(* IEC 61131-3 sources: RL_MAR/experiments/results/ablation/Ablation_single_agent_deepseek-ai_DeepSeek-V3.2_20260603_033757, 94 files *)

(* ---- hard_92.st ---- *)
FUNCTION_BLOCK FB_BreakerControlSystem
VAR_INPUT
    B10_1_Trip : BOOL;
    B10_1_Close : BOOL;
    B10_2_Trip : BOOL;
    B10_2_Close : BOOL;
    B10_12_Trip : BOOL;
    B10_12_Close : BOOL;
    B54_Trip : BOOL;
    B54_Close : BOOL;
    B55_Trip : BOOL;
    B55_Close : BOOL;
    B56_Trip : BOOL;
    B56_Close : BOOL;
    B57_Trip : BOOL;
    B57_Close : BOOL;
END_VAR

VAR_OUTPUT
    Point_1a : INT;
    Point_2a : INT;
    Point_3a : INT;
    Point_4a : INT;
    B10_1_Opened : BOOL;
    B10_1_Closed : BOOL;
    B10_2_Opened : BOOL;
    B10_2_Closed : BOOL;
    B10_12_Opened : BOOL;
    B10_12_Closed : BOOL;
    B54_Opened : BOOL;
    B54_Closed : BOOL;
    B55_Opened : BOOL;
    B55_Closed : BOOL;
    B56_Opened : BOOL;
    B56_Closed : BOOL;
    B57_Opened : BOOL;
    B57_Closed : BOOL;
END_VAR

VAR
    SEL86_OUT : INT;
    MOVE89_OUT : INT;
    SEL66_OUT : INT;
    MOVE69_OUT : INT;
    SEL96_OUT : INT;
    MOVE99_OUT : INT;
    SEL106_OUT : INT;
    MOVE109_OUT : INT;
END_VAR

(* Breaker State Transition Logic *)
(* B10_1 State Management *)
IF B10_1_Close THEN
    B10_1_Closed := TRUE;
    B10_1_Opened := FALSE;
ELSIF B10_1_Trip THEN
    B10_1_Closed := FALSE;
    B10_1_Opened := TRUE;
END_IF;

(* B10_2 State Management *)
IF B10_2_Close THEN
    B10_2_Closed := TRUE;
    B10_2_Opened := FALSE;
ELSIF B10_2_Trip THEN
    B10_2_Closed := FALSE;
    B10_2_Opened := TRUE;
END_IF;

(* B10_12 State Management *)
IF B10_12_Close THEN
    B10_12_Closed := TRUE;
    B10_12_Opened := FALSE;
ELSIF B10_12_Trip THEN
    B10_12_Closed := FALSE;
    B10_12_Opened := TRUE;
END_IF;

(* B54 State Management *)
IF B54_Close THEN
    B54_Closed := TRUE;
    B54_Opened := FALSE;
ELSIF B54_Trip THEN
    B54_Closed := FALSE;
    B54_Opened := TRUE;
END_IF;

(* B55 State Management *)
IF B55_Close THEN
    B55_Closed := TRUE;
    B55_Opened := FALSE;
ELSIF B55_Trip THEN
    B55_Closed := FALSE;
    B55_Opened := TRUE;
END_IF;

(* B56 State Management *)
IF B56_Close THEN
    B56_Closed := TRUE;
    B56_Opened := FALSE;
ELSIF B56_Trip THEN
    B56_Closed := FALSE;
    B56_Opened := TRUE;
END_IF;

(* B57 State Management *)
IF B57_Close THEN
    B57_Closed := TRUE;
    B57_Opened := FALSE;
ELSIF B57_Trip THEN
    B57_Closed := FALSE;
    B57_Opened := TRUE;
END_IF;

(* Point_1a Calculation *)
IF B54_Closed AND ((B10_12_Closed AND B10_1_Closed) OR B10_2_Closed) THEN
    Point_1a := 0;
ELSE
    Point_1a := 138;
END_IF;

(* Point_2a Calculation *)
IF B55_Closed AND ((B10_12_Closed AND B10_1_Closed) OR B10_2_Closed) THEN
    Point_2a := 0;
ELSE
    Point_2a := 138;
END_IF;

(* Point_3a Calculation *)
IF B56_Closed AND ((B10_12_Closed AND B10_2_Closed) OR B10_1_Closed) THEN
    Point_3a := 0;
ELSE
    Point_3a := 138;
END_IF;

(* Point_4a Calculation *)
IF B57_Closed AND ((B10_12_Closed AND B10_2_Closed) OR B10_1_Closed) THEN
    Point_4a := 0;
ELSE
    Point_4a := 138;
END_IF;

END_FUNCTION_BLOCK

(* ---- hard_93.st ---- *)
FUNCTION_BLOCK FB_CircuitControl
VAR_INPUT
    Reset_All_CB : BOOL;
    Current_Fault_on_TRSF1 : INT;
    Current_Fault_on_66BUS1 : INT;
END_VAR

VAR_OUTPUT
    Short_Circuit_TRSF1 : BOOL;
    Short_Circuit_66BUS : BOOL;
    Open_CB1_66KV : BOOL;
    Open_CB2_66KV : BOOL;
    Open_CB_TRSF1 : BOOL;
    Open_CB2_22KV : BOOL;
END_VAR

VAR
    Threshold500 : INT := 500;
    Prev_Open_CB2_22KV : BOOL;
    Prev_Open_CB1_66KV : BOOL;
    Prev_Open_CB_TRSF1 : BOOL;
    Temp_Open_CB2_22KV : BOOL;
    Temp_Open_CB1_66KV : BOOL;
    Temp_Open_CB_TRSF1 : BOOL;
END_VAR

(* Short Circuit Detection *)
Short_Circuit_66BUS := (Current_Fault_on_66BUS1 > Threshold500);
Short_Circuit_TRSF1 := (Current_Fault_on_TRSF1 > Threshold500);

(* Save previous states for edge detection and logic *)
Prev_Open_CB2_22KV := Open_CB2_22KV;
Prev_Open_CB1_66KV := Open_CB1_66KV;
Prev_Open_CB_TRSF1 := Open_CB_TRSF1;

(* Initial Reset Condition *)
IF Reset_All_CB THEN
    Open_CB2_22KV := FALSE;
    Open_CB1_66KV := FALSE;
    Open_CB_TRSF1 := FALSE;
    Open_CB2_66KV := TRUE;
    RETURN;
END_IF;

(* Step 1: Initial Open_CB2_22KV Logic *)
Temp_Open_CB2_22KV := FALSE;
IF (Prev_Open_CB2_22KV = FALSE) THEN
    IF ((Open_CB1_66KV AND Open_CB_TRSF1) OR Short_Circuit_66BUS) THEN
        Temp_Open_CB2_22KV := TRUE;
    END_IF;
END_IF;

(* Step 2: Initial Open_CB1_66KV Logic *)
Temp_Open_CB1_66KV := FALSE;
IF (Temp_Open_CB2_22KV = FALSE) THEN
    IF ((Prev_Open_CB1_66KV AND Open_CB_TRSF1) OR Short_Circuit_66BUS) THEN
        Temp_Open_CB1_66KV := TRUE;
    END_IF;
END_IF;

(* Step 3: Initial Open_CB_TRSF1 Logic *)
Temp_Open_CB_TRSF1 := FALSE;
IF (Temp_Open_CB2_22KV = FALSE) THEN
    IF ((Open_CB1_66KV AND Prev_Open_CB_TRSF1) OR Short_Circuit_66BUS) THEN
        Temp_Open_CB_TRSF1 := TRUE;
    END_IF;
END_IF;

(* Step 4: Open_CB2_66KV is always TRUE *)
Open_CB2_66KV := TRUE;

(* Step 5: Update Open_CB2_22KV again *)
IF (Prev_Open_CB2_22KV = FALSE) THEN
    IF ((Open_CB2_66KV AND Open_CB1_66KV AND Open_CB_TRSF1) OR Short_Circuit_TRSF1) THEN
        Temp_Open_CB2_22KV := TRUE;
    END_IF;
END_IF;

(* Step 6: Update Open_CB1_66KV again *)
IF (Temp_Open_CB2_22KV = FALSE) THEN
    IF ((Open_CB2_66KV AND Prev_Open_CB1_66KV AND Open_CB_TRSF1) OR Short_Circuit_TRSF1) THEN
        Temp_Open_CB1_66KV := TRUE;
    END_IF;
END_IF;

(* Step 7: Update Open_CB_TRSF1 again *)
IF (Temp_Open_CB2_22KV = FALSE) THEN
    IF ((Open_CB2_66KV AND Open_CB1_66KV AND Prev_Open_CB_TRSF1) OR Short_Circuit_TRSF1) THEN
        Temp_Open_CB_TRSF1 := TRUE;
    END_IF;
END_IF;

(* Apply final values with anti-rapid switching: only change if new state is TRUE and current is FALSE *)
IF (Temp_Open_CB2_22KV AND (NOT Open_CB2_22KV)) THEN
    Open_CB2_22KV := TRUE;
END_IF;

IF (Temp_Open_CB1_66KV AND (NOT Open_CB1_66KV)) THEN
    Open_CB1_66KV := TRUE;
END_IF;

IF (Temp_Open_CB_TRSF1 AND (NOT Open_CB_TRSF1)) THEN
    Open_CB_TRSF1 := TRUE;
END_IF;

END_FUNCTION_BLOCK

(* ---- hard_94.st ---- *)
FUNCTION_BLOCK FB_AdvancedCircuitBreakerControl
VAR_INPUT
    S_AL1_P_B1 : BOOL;
    S_AL1_P_B2 : BOOL;
    S_AL1_MCB : BOOL;
    MCB_BUSY : BOOL;
    MCB_ERROR : BOOL;
    S_AL1_MCBR : BOOL;
    MCBR_BUSY : BOOL;
    MCBR_ERROR : BOOL;
    S_AL1_P_B3 : BOOL;
    S_AL1_MCB2 : BOOL;
    S_AL1_MCBR2 : BOOL;
END_VAR

VAR_OUTPUT
    E_AL1_B1 : BOOL;
    PUWS_AL1_B1_PLUS : BOOL;
    PUWS_AL1_B1_RIGHT : BOOL;
    PAS_AL1_PLUS : BOOL;
    PAS_AL1_TURN : BOOL;
END_VAR

VAR
    PPAL1 : BOOL := TRUE;
    PP0 : BOOL := TRUE;
    PP1 : BOOL := FALSE;
    PP2 : BOOL := FALSE;
    PP3 : BOOL := FALSE;
    PP4 : BOOL := FALSE;
    MCB : BOOL := TRUE;
    PP5 : BOOL := FALSE;
    PP7 : BOOL := FALSE;
    PPL3 : BOOL := FALSE;
    PPL4 : BOOL := FALSE;
    MCBR : BOOL := TRUE;
    PPL5 : BOOL := FALSE;
    PPL7 : BOOL := FALSE;
    STABLE : BOOL := FALSE;
    MCB_CONTROL : BOOL;
END_VAR

METHOD Main : BOOL
VAR_INST
END_VAR

STABLE := FALSE;

WHILE (STABLE = FALSE) DO
    STABLE := TRUE;

    // PP0 to PP1
    IF (PP0 = TRUE) AND (NOT MCB_CONTROL) AND (PP1 = FALSE) THEN
        PP0 := FALSE;
        PP1 := TRUE;
        STABLE := FALSE;
    END_IF;

    // PP1 to PP2
    IF (PP1 = TRUE) AND S_AL1_P_B1 AND (PP2 = FALSE) THEN
        PP1 := FALSE;
        PP2 := TRUE;
        STABLE := FALSE;
    END_IF;

    // PP2 to PP3
    IF (PP2 = TRUE) AND S_AL1_P_B2 AND (NOT MCB_CONTROL) AND (PP3 = FALSE) THEN
        PP2 := FALSE;
        PP3 := TRUE;
        STABLE := FALSE;
    END_IF;

    // PP3 to PP4
    IF (PP3 = TRUE) AND S_AL1_MCB AND (PP4 = FALSE) AND (PP1 = FALSE) THEN
        PP3 := FALSE;
        PP4 := TRUE;
        PP1 := TRUE;
        STABLE := FALSE;
    END_IF;

    // PP4 to PP5
    IF (PP4 = TRUE) AND (MCB = TRUE) AND MCB_BUSY AND (PP5 = FALSE) THEN
        PP4 := FALSE;
        MCB := FALSE;
        PP5 := TRUE;
        STABLE := FALSE;
    END_IF;

    // PP5 to PP7
    IF (PP5 = TRUE) AND S_AL1_MCB2 AND (PP7 = FALSE) AND (MCB = FALSE) THEN
        PP5 := FALSE;
        PP7 := TRUE;
        MCB := TRUE;
        STABLE := FALSE;
    END_IF;

    // PP7 to End
    IF (PP7 = TRUE) AND S_AL1_P_B3 THEN
        PP7 := FALSE;
        STABLE := FALSE;
    END_IF;

    // PP2 to PPL3
    IF (PP2 = TRUE) AND S_AL1_P_B2 AND MCB_CONTROL AND (PPL3 = FALSE) AND (PP1 = FALSE) THEN
        PP2 := FALSE;
        PPL3 := TRUE;
        PP1 := TRUE;
        STABLE := FALSE;
    END_IF;

    // PPL3 to PPL4
    IF (PPL3 = TRUE) AND S_AL1_MCBR AND (PPL4 = FALSE) THEN
        PPL3 := FALSE;
        PPL4 := TRUE;
        STABLE := FALSE;
    END_IF;

    // PPL4 to PPL5
    IF (PPL4 = TRUE) AND (MCBR = TRUE) AND MCBR_BUSY AND (PPL5 = FALSE) THEN
        PPL4 := FALSE;
        MCBR := FALSE;
        PPL5 := TRUE;
        STABLE := FALSE;
    END_IF;

    // PPL5 to PPL7
    IF (PPL5 = TRUE) AND S_AL1_MCBR2 AND (PPL7 = FALSE) AND (MCBR = FALSE) THEN
        PPL5 := FALSE;
        PPL7 := TRUE;
        MCBR := TRUE;
        STABLE := FALSE;
    END_IF;

    // PPL7 to End
    IF (PPL7 = TRUE) AND S_AL1_P_B3 THEN
        PPL7 := FALSE;
        STABLE := FALSE;
    END_IF;
END_WHILE;

// Output Control
// Set outputs based on active states
IF (PP0 = TRUE) OR (PP1 = TRUE) THEN
    E_AL1_B1 := TRUE;
ELSE
    E_AL1_B1 := FALSE;
END_IF;

IF (PP3 = TRUE) THEN
    MCB_CONTROL := TRUE;
ELSE
    MCB_CONTROL := FALSE;
END_IF;

IF (PPL3 = TRUE) OR (PPL4 = TRUE) THEN
    PAS_AL1_PLUS := TRUE;
    PAS_AL1_TURN := TRUE;
ELSE
    PAS_AL1_PLUS := FALSE;
    PAS_AL1_TURN := FALSE;
END_IF;

IF (PPAL1 = TRUE) OR (PP2 = TRUE) THEN
    PUWS_AL1_B1_PLUS := TRUE;
ELSE
    PUWS_AL1_B1_PLUS := FALSE;
END_IF;

IF (PP2 = TRUE) OR (PP3 = TRUE) OR (PPL3 = TRUE) THEN
    E_AL1_B1 := FALSE;
END_IF;

IF (PP0 = TRUE) OR (PP3 = TRUE) THEN
    MCB_CONTROL := FALSE;
END_IF;

IF (PP0 = TRUE) OR (PP3 = TRUE) OR (PP4 = TRUE) THEN
    PAS_AL1_PLUS := FALSE;
    PAS_AL1_TURN := FALSE;
END_IF;

IF (PPAL1 = TRUE) OR (PP2 = TRUE) THEN
    PUWS_AL1_B1_RIGHT := FALSE;
END_IF;

Main := TRUE;
END_METHOD

END_FUNCTION_BLOCK

(* ---- hf_1.st ---- *)
FUNCTION_BLOCK StackMin
VAR_INPUT
    push : BOOL;
    pop : BOOL;
    reset : BOOL;
END_VAR
VAR_OUTPUT
    error : BOOL;
    status : WORD;
END_VAR
VAR_IN_OUT
    item : INT;
    stack : ARRAY[0..3] OF INT;
END_VAR
VAR
    top : INT := -1;
    i : INT;
    minIndex : INT;
    minValue : INT;
END_VAR

// Reset has highest priority
IF reset THEN
    top := -1;
    error := FALSE;
    status := 16#0000;

// Push operation (prioritized over pop if both are active)
ELSIF push THEN
    IF top >= 3 THEN
        error := TRUE;
        status := 16#8A04;
    ELSE
        top := top + 1;
        stack[top] := item;
        error := FALSE;
        status := 16#0000;
    END_IF;

// Pop operation (only if push is not active)
ELSIF pop THEN
    IF top < 0 THEN
        error := TRUE;
        status := 16#8A05;
    ELSE
        // Find minimum value and its index
        minIndex := 0;
        minValue := stack[0];
        i := 1;
        WHILE i <= top DO
            IF stack[i] < minValue THEN
                minValue := stack[i];
                minIndex := i;
            END_IF;
            i := i + 1;
        END_WHILE;

        // Return minimum value
        item := minValue;

        // Shift elements down to remove the minimum
        i := minIndex;
        WHILE i < top DO
            stack[i] := stack[i + 1];
            i := i + 1;
        END_WHILE;

        // Clear the vacated position (optional but clean)
        stack[top] := 0;

        // Update top index
        top := top - 1;

        error := FALSE;
        status := 16#0000;
    END_IF;

// No operation
ELSE
    error := FALSE;
    status := 16#0000;
END_IF;

END_FUNCTION_BLOCK

(* ---- hf_10.st ---- *)
FUNCTION_BLOCK FloatingAverage
VAR_INPUT
    cyclicExecution : BOOL;
    trigger : BOOL;
    value : REAL;
    windowSize : INT;
    reset : BOOL;
END_VAR

VAR_OUTPUT
    average : REAL;
    windowSizeReached : BOOL;
    error : BOOL;
    status : WORD;
END_VAR

VAR
    dataBuffer : ARRAY[1..100] OF REAL; (* Buffer to store the data values *)
    bufferIndex : INT := 1; (* Index to track the current position in the buffer *)
    sum : REAL := 0.0; (* Sum of the data values in the buffer *)
    currentWindowSize : INT := 0; (* Current number of valid data points in buffer *)
    triggerPrev : BOOL := FALSE; (* Previous trigger state for edge detection *)
END_VAR

(* Main execution logic *)
IF reset THEN
    (* Reset all internal states *)
    bufferIndex := 1;
    sum := 0.0;
    currentWindowSize := 0;
    average := 0.0;
    windowSizeReached := FALSE;
    error := FALSE;
    status := 16#0000;

    (* Clear buffer *)
    FOR i := 1 TO 100 DO
        dataBuffer[i] := 0.0;
    END_FOR;

ELSIF windowSize < 1 OR windowSize > 100 THEN
    (* Window size error *)
    error := TRUE;
    status := 16#8200;
    windowSizeReached := FALSE;

ELSE
    (* Check if we should process new data *)
    IF cyclicExecution OR (trigger AND NOT triggerPrev) THEN
        (* Update buffer with new value *)
        dataBuffer[bufferIndex] := value;

        (* Update sum - remove oldest value if window is full *)
        IF currentWindowSize < windowSize THEN
            (* Window not yet full, just add new value *)
            sum := sum + value;
            currentWindowSize := currentWindowSize + 1;
        ELSE
            (* Window is full, replace oldest value *)
            sum := sum - dataBuffer[bufferIndex] + value;
        END_IF;

        (* Update buffer index with wrap-around *)
        bufferIndex := bufferIndex + 1;
        IF bufferIndex > windowSize THEN
            bufferIndex := 1;
        END_IF;

        (* Calculate average *)
        IF currentWindowSize > 0 THEN
            average := sum / currentWindowSize;
        ELSE
            average := 0.0;
        END_IF;

        (* Update windowSizeReached flag *)
        windowSizeReached := (currentWindowSize >= windowSize);

        (* Clear error and set success status *)
        error := FALSE;
        status := 16#0000;
    END_IF;

    (* Update trigger previous state for edge detection *)
    triggerPrev := trigger;
END_IF;

(* Ensure outputs are valid even when no new data is processed *)
IF NOT (cyclicExecution OR (trigger AND NOT triggerPrev)) AND NOT reset THEN
    (* Maintain current outputs when not processing new data *)
    IF currentWindowSize > 0 THEN
        average := sum / currentWindowSize;
    ELSE
        average := 0.0;
    END_IF;
    windowSizeReached := (currentWindowSize >= windowSize);
END_IF;

END_FUNCTION_BLOCK

(* ---- hf_11.st ---- *)
FUNCTION_BLOCK FB_BottleProcessing
VAR_INPUT
    bottleSensor : BOOL;
    cleaningConfirmButton : BOOL;
    fillingConfirmButton : BOOL;
    cappingConfirmButton : BOOL;
    packingConfirmButton : BOOL;
    finishedButton : BOOL;
END_VAR

VAR_OUTPUT
    Pump_Motor : BOOL;
    Filling_Valve : BOOL;
    Capping_Machine : BOOL;
    Packing_Machine : BOOL;
    Completion_Light : BOOL;
END_VAR

VAR
    State : INT := 0; (* 0=Waiting, 1=Cleaning, 2=Filling, 3=Capping, 4=Packing, 5=Completed *)
END_VAR

CASE State OF
    0: (* Waiting state *)
        IF bottleSensor THEN
            Pump_Motor := TRUE;
            State := 1;
        END_IF;

    1: (* Cleaning state *)
        IF cleaningConfirmButton THEN
            Pump_Motor := FALSE;
            Filling_Valve := TRUE;
            State := 2;
        END_IF;

    2: (* Filling state *)
        IF fillingConfirmButton THEN
            Filling_Valve := FALSE;
            Capping_Machine := TRUE;
            State := 3;
        END_IF;

    3: (* Capping state *)
        IF cappingConfirmButton THEN
            Capping_Machine := FALSE;
            Packing_Machine := TRUE;
            State := 4;
        END_IF;

    4: (* Packing state *)
        IF packingConfirmButton THEN
            Packing_Machine := FALSE;
            Completion_Light := TRUE;
            State := 5;
        END_IF;

    5: (* Completed state *)
        IF finishedButton THEN
            Completion_Light := FALSE;
            Pump_Motor := FALSE;
            Filling_Valve := FALSE;
            Capping_Machine := FALSE;
            Packing_Machine := FALSE;
            State := 0;
        END_IF;
END_CASE;
END_FUNCTION_BLOCK

(* ---- hf_12.st ---- *)
FUNCTION_BLOCK MaterialMixing
VAR_INPUT
    estop : BOOL; (* Emergency Stop Signal, FALSE: Emergency stop triggered, TRUE: No emergency stop triggered *)
    opeMode : BOOL; (* Operation Mode, FALSE: Manual Operation Mode, TRUE: Automatic Operation Mode *)
    valveAStart : BOOL; (* Valve A Start Button *)
    valveBStart : BOOL; (* Valve B Start Button *)
    valveCStart : BOOL; (* Valve C Start Button *)
    valveDStart : BOOL; (* Valve D Start Button *)
    mixMotorStart : BOOL; (* Mixing Motor Start Button *)
    autoStart : BOOL; (* Automatic Start Button *)
    processMode : BOOL; (* Process Mode *)
    levelSensor : INT; (* Liquid Level Sensor, unit cm *)
    mixMotorComplete : BOOL; (* Mixing Complete Signal *)
END_VAR
VAR_OUTPUT
    valveARun : BOOL; (* Valve A Run Command *)
    valveBRun : BOOL; (* Valve B Run Command *)
    valveCRun : BOOL; (* Valve C Run Command *)
    valveDRun : BOOL; (* Valve D Run Command *)
    mixMotorRun : BOOL; (* Mixing Motor Run Command *)
END_VAR
VAR
    (* Edge detection variables for manual mode *)
    prevValveAStart : BOOL := FALSE;
    prevValveBStart : BOOL := FALSE;
    prevValveCStart : BOOL := FALSE;
    prevValveDStart : BOOL := FALSE;
    prevMixMotorStart : BOOL := FALSE;
    prevAutoStart : BOOL := FALSE;

    (* Automatic mode state variables *)
    autoActive : BOOL := FALSE;
    autoStep : INT := 0;
END_VAR

(* Emergency stop logic - highest priority *)
IF NOT estop THEN
    (* Emergency stop triggered - stop all equipment *)
    valveARun := FALSE;
    valveBRun := FALSE;
    valveCRun := FALSE;
    valveDRun := FALSE;
    mixMotorRun := FALSE;
    autoActive := FALSE;
    autoStep := 0;
ELSE
    (* Normal operation *)
    IF opeMode THEN
        (* Automatic Mode *)

        (* Toggle automatic process on rising edge of autoStart *)
        IF autoStart AND NOT prevAutoStart THEN
            autoActive := NOT autoActive;
            IF autoActive THEN
                autoStep := 1; (* Start with step 1: open valve A *)
            ELSE
                autoStep := 0; (* Reset to idle *)
            END_IF;
        END_IF;
        prevAutoStart := autoStart;

        (* Automatic process state machine *)
        IF autoActive THEN
            CASE autoStep OF
                1: (* Step 1: Open valve A *)
                    valveARun := TRUE;
                    valveBRun := FALSE;
                    valveCRun := FALSE;
                    valveDRun := FALSE;
                    mixMotorRun := FALSE;

                    IF levelSensor >= 50 THEN
                        valveARun := FALSE;
                        autoStep := 2; (* Move to step 2: open valve B *)
                    END_IF;

                2: (* Step 2: Open valve B *)
                    valveBRun := TRUE;

                    IF levelSensor >= 80 THEN
                        valveBRun := FALSE;
                        IF processMode THEN
                            autoStep := 3; (* ProcessMode = TRUE: go to step 3 *)
                        ELSE
                            autoStep := 4; (* ProcessMode = FALSE: skip to step 4 *)
                        END_IF;
                    END_IF;

                3: (* Step 3: Open valve C (only when processMode = TRUE) *)
                    valveCRun := TRUE;

                    IF levelSensor >= 100 THEN
                        valveCRun := FALSE;
                        autoStep := 4; (* Move to step 4: start mixing *)
                    END_IF;

                4: (* Step 4: Start mixing motor *)
                    mixMotorRun := TRUE;

                    IF mixMotorComplete THEN
                        mixMotorRun := FALSE;
                        autoStep := 5; (* Move to step 5: open valve D *)
                    END_IF;

                5: (* Step 5: Open valve D and end process *)
                    valveDRun := TRUE;
                    autoActive := FALSE; (* Process complete *)
                    autoStep := 0; (* Reset state machine *)

            END_CASE;
        ELSE
            (* Automatic mode inactive - ensure all outputs are off *)
            valveARun := FALSE;
            valveBRun := FALSE;
            valveCRun := FALSE;
            valveDRun := FALSE;
            mixMotorRun := FALSE;
        END_IF;

    ELSE
        (* Manual Mode *)

        (* Valve A toggle on rising edge *)
        IF valveAStart AND NOT prevValveAStart THEN
            valveARun := NOT valveARun;
        END_IF;
        prevValveAStart := valveAStart;

        (* Valve B toggle on rising edge *)
        IF valveBStart AND NOT prevValveBStart THEN
            valveBRun := NOT valveBRun;
        END_IF;
        prevValveBStart := valveBStart;

        (* Valve C toggle on rising edge *)
        IF valveCStart AND NOT prevValveCStart THEN
            valveCRun := NOT valveCRun;
        END_IF;
        prevValveCStart := valveCStart;

        (* Valve D toggle on rising edge *)
        IF valveDStart AND NOT prevValveDStart THEN
            valveDRun := NOT valveDRun;
        END_IF;
        prevValveDStart := valveDStart;

        (* Mixing motor toggle on rising edge *)
        IF mixMotorStart AND NOT prevMixMotorStart THEN
            mixMotorRun := NOT mixMotorRun;
        END_IF;
        prevMixMotorStart := mixMotorStart;

    END_IF;
END_IF;

END_FUNCTION_BLOCK

(* ---- hf_13.st ---- *)
FUNCTION_BLOCK TON
VAR_INPUT
    IN : BOOL;
    PT : DINT;
    CYCLE_TIME : DINT;
END_VAR
VAR_OUTPUT
    Q : BOOL;
    ET : DINT;
END_VAR
VAR
    elapsedTimeInternal : DINT := 0;
    IN_PREV : BOOL := FALSE;
END_VAR

IF IN THEN
    IF NOT IN_PREV THEN
        elapsedTimeInternal := 0;
    END_IF;

    IF elapsedTimeInternal < PT THEN
        elapsedTimeInternal := elapsedTimeInternal + CYCLE_TIME;
        Q := FALSE;
    ELSE
        elapsedTimeInternal := PT;
        Q := TRUE;
    END_IF;

    ET := elapsedTimeInternal;
ELSE
    Q := FALSE;
    ET := 0;
    elapsedTimeInternal := 0;
END_IF;
IN_PREV := IN;
END_FUNCTION_BLOCK

FUNCTION_BLOCK LightsControl
VAR_INPUT
    button1 : BOOL; (* Button 1: Automatic/Manual Mode Select *)
    button2 : BOOL; (* Button 2: Manual Control/Green Light Req *)
    button3 : BOOL; (* Button 3: Manual Control/Red Light Req *)
    CYCLE_TIME : DINT; (* Time elapsed in current cycle (in ms) *)
END_VAR
VAR_OUTPUT
    greenLight : BOOL; (* Green light *)
    redLight : BOOL; (* Red light *)
    yellowLight : BOOL; (* Yellow light *)
END_VAR
VAR
    (* Timers for control *)
    timerAuto : TON;
    timerGreen : TON;
    timerRed : TON;
    timerYellow : TON;

    currentState : INT := 0;
    autoRunTimer : BOOL;

    (* Internal variables for manual mode *)
    manualGreenActive : BOOL;
    manualRedActive : BOOL;
    manualYellowActive : BOOL;
END_VAR

(* Reset manual timers at start of every cycle as required *)
timerGreen(IN := FALSE, PT := 1000, CYCLE_TIME := CYCLE_TIME);
timerRed(IN := FALSE, PT := 2000, CYCLE_TIME := CYCLE_TIME);
timerYellow(IN := FALSE, PT := 1000, CYCLE_TIME := CYCLE_TIME);

(* Determine manual mode activation *)
manualGreenActive := button2 AND NOT button3;
manualRedActive := button2 AND NOT button3;
manualYellowActive := NOT button2 AND button3;

(* Automatic Mode *)
IF button1 THEN
    autoRunTimer := TRUE;
    timerAuto(IN := autoRunTimer, PT := 1000, CYCLE_TIME := CYCLE_TIME);

    CASE currentState OF
        0: (* State 0: Green light on for 1 second *)
            greenLight := TRUE;
            redLight := FALSE;
            yellowLight := FALSE;
            IF timerAuto.Q THEN
                currentState := 1;
                timerAuto.IN := FALSE; (* Reset timer *)
            END_IF;

        1: (* State 1: Red light on for 1 second *)
            greenLight := FALSE;
            redLight := TRUE;
            yellowLight := FALSE;
            IF timerAuto.Q THEN
                currentState := 2;
                timerAuto.IN := FALSE; (* Reset timer *)
            END_IF;

        2: (* State 2: Yellow light on for 1 second *)
            greenLight := FALSE;
            redLight := FALSE;
            yellowLight := TRUE;
            IF timerAuto.Q THEN
                currentState := 0;
                timerAuto.IN := FALSE; (* Reset timer *)
            END_IF;
    END_CASE;

(* Manual Mode *)
ELSE
    autoRunTimer := FALSE;
    timerAuto.IN := FALSE;
    currentState := 0;

    (* Activate timers based on button combinations *)
    IF manualGreenActive THEN
        timerGreen(IN := TRUE, PT := 1000, CYCLE_TIME := CYCLE_TIME);
        timerRed(IN := TRUE, PT := 2000, CYCLE_TIME := CYCLE_TIME);
    ELSIF manualYellowActive THEN
        timerYellow(IN := TRUE, PT := 1000, CYCLE_TIME := CYCLE_TIME);
    ELSIF button2 AND button3 THEN
        timerGreen(IN := TRUE, PT := 1000, CYCLE_TIME := CYCLE_TIME);
    END_IF;

    (* Manual mode logic *)
    IF NOT button2 AND NOT button3 THEN
        (* Both FALSE: All lights off *)
        greenLight := FALSE;
        redLight := FALSE;
        yellowLight := FALSE;

    ELSIF button2 AND NOT button3 THEN
        (* button2 TRUE, button3 FALSE *)
        greenLight := TRUE;
        redLight := timerRed.Q; (* Blinks at 0.5Hz (2000ms period) *)
        yellowLight := FALSE;

    ELSIF NOT button2 AND button3 THEN
        (* button2 FALSE, button3 TRUE *)
        greenLight := FALSE;
        redLight := TRUE;
        yellowLight := NOT timerYellow.Q; (* Blinks at 1Hz (1000ms period) *)

    ELSIF button2 AND button3 THEN
        (* Both TRUE *)
        greenLight := NOT timerGreen.Q; (* Blinks at 1Hz (1000ms period) *)
        redLight := FALSE;
        yellowLight := TRUE;
    END_IF;
END_IF;
END_FUNCTION_BLOCK

(* ---- hf_14.st ---- *)
FUNCTION_BLOCK TruckGarage
VAR_INPUT
    enter_flag : BOOL;
    exit_flag : BOOL;
    VehicleNumber_in : INT;
END_VAR
VAR_OUTPUT
    truck_row : INT;
    truck_col : INT;
    truck_VehicleNumber : INT;
END_VAR
VAR_IN_OUT
    garage : ARRAY[1..3, 1..5] OF STRUCT
        Occupied : BOOL;
        VehicleNumber : INT;
    END_STRUCT;
END_VAR
VAR
    i : INT;
    j : INT;
    found : BOOL;
END_VAR

// Entry logic
IF enter_flag THEN
    found := FALSE;

    // Search from last row to first, last column to first
    FOR i := 3 TO 1 BY -1 DO
        FOR j := 5 TO 1 BY -1 DO
            IF NOT garage[i, j].Occupied AND NOT found THEN
                // Found empty spot
                garage[i, j].Occupied := TRUE;
                garage[i, j].VehicleNumber := VehicleNumber_in;
                found := TRUE;
            END_IF
        END_FOR
    END_FOR
END_IF

// Exit logic
IF exit_flag THEN
    found := FALSE;

    // Search from first row to last, first column to last
    FOR i := 1 TO 3 DO
        FOR j := 1 TO 5 DO
            IF garage[i, j].Occupied AND garage[i, j].VehicleNumber = VehicleNumber_in AND NOT found THEN
                // Found vehicle to exit
                truck_row := i;
                truck_col := j;
                truck_VehicleNumber := garage[i, j].VehicleNumber;

                // Clear the parking spot
                garage[i, j].Occupied := FALSE;
                garage[i, j].VehicleNumber := 0;
                found := TRUE;
            END_IF
        END_FOR
    END_FOR

    // If vehicle not found, clear output
    IF NOT found THEN
        truck_row := 0;
        truck_col := 0;
        truck_VehicleNumber := 0;
    END_IF
END_IF

// Clear outputs when no operation
IF NOT enter_flag AND NOT exit_flag THEN
    truck_row := 0;
    truck_col := 0;
    truck_VehicleNumber := 0;
END_IF
END_FUNCTION_BLOCK

(* ---- hf_15.st ---- *)
FUNCTION_BLOCK FB_MergeBytes
VAR_INPUT
    byteArray : ARRAY[1..20] OF DINT; (* Byte array to be merged *)
END_VAR
VAR_OUTPUT
    dwordArray : ARRAY[1..10] OF DINT; (* Merged double word array *)
    mergeDwordNum : DINT;
END_VAR
VAR
    i, j : DINT;
    tempDword : DWORD;
    bytePos : DINT;
    dwordPos : DINT;
    maxDwords : DINT;
END_VAR
VAR CONSTANT
    BYTE_ARRAY_SIZE : DINT := 20; (* Size of the input byte array *)
    DWORD_ARRAY_SIZE : DINT := 10; (* Size of the output DINT array *)
END_VAR

BEGIN
    mergeDwordNum := 0;

    (* Clear output array *)
    FOR i := 1 TO DWORD_ARRAY_SIZE DO
        dwordArray[i] := 0;
    END_FOR;

    (* Calculate maximum number of DWORDs we can merge *)
    maxDwords := MIN(BYTE_ARRAY_SIZE / 4, DWORD_ARRAY_SIZE);

    (* Merge bytes into DWORDs *)
    FOR dwordPos := 0 TO maxDwords - 1 DO
        tempDword := 0;
        bytePos := dwordPos * 4;

        (* Check if we have enough bytes remaining *)
        IF (bytePos + 4) <= BYTE_ARRAY_SIZE THEN
            (* Merge 4 bytes into 1 DWORD *)
            FOR j := 0 TO 3 DO
                (* Shift each byte into position and combine *)
                tempDword := tempDword OR (SHL(TO_DWORD(byteArray[bytePos + j + 1] AND 16#FF), (3 - j) * 8));
            END_FOR;

            (* Store the merged DWORD *)
            dwordArray[dwordPos + 1] := TO_DINT(tempDword);
            mergeDwordNum := mergeDwordNum + 1;
        END_IF;
    END_FOR;

END_FUNCTION_BLOCK

(* ---- hf_16.st ---- *)
FUNCTION_BLOCK FB_LinearizeValue
VAR_INPUT
    InputValue : REAL; // Floating point input, raw measurement value
END_VAR

VAR_OUTPUT
    LinearizedValue : REAL; // Converted linear value
    Error : BOOL; // Error status indicator
    Status : WORD; // Status code
END_VAR

VAR
    // No additional variables needed here
END_VAR

// Main execution logic
IF InputValue < 1200.0 THEN
    // Below minimum range
    LinearizedValue := 150.0;
    Error := TRUE;
    Status := 16#8001;
ELSIF InputValue >= 1200.0 AND InputValue < 3600.0 THEN
    // Range 1: 1200 to 3600
    LinearizedValue := 150.0 + (InputValue - 1200.0) * (240.0 - 150.0) / (3600.0 - 1200.0);
    Error := FALSE;
    Status := 16#0000;
ELSIF InputValue >= 3600.0 AND InputValue < 4800.0 THEN
    // Range 2: 3600 to 4800
    LinearizedValue := 240.0 + (InputValue - 3600.0) * (560.0 - 240.0) / (4800.0 - 3600.0);
    Error := FALSE;
    Status := 16#0000;
ELSIF InputValue >= 4800.0 AND InputValue <= 7000.0 THEN
    // Range 3: 4800 to 7000
    LinearizedValue := 560.0 + (InputValue - 4800.0) * (720.0 - 560.0) / (7000.0 - 4800.0);
    Error := FALSE;
    Status := 16#0000;
ELSE
    // Above maximum range
    LinearizedValue := 720.0;
    Error := TRUE;
    Status := 16#8001;
END_IF;

END_FUNCTION_BLOCK

(* ---- hf_17.st ---- *)
FUNCTION_BLOCK FB_WarehouseManagement
VAR_INPUT
    requestIn : BOOL := FALSE;
    requestOut : BOOL := FALSE;
END_VAR

VAR_OUTPUT
    productNum : INT := 0;
    libFreeNum : INT := 9;
    error : BOOL := FALSE;
    status : WORD := 16#0000;
END_VAR

VAR_IN_OUT
    library : ARRAY[1..9] OF BOOL;
END_VAR

VAR
    i : INT;
    found : BOOL;
    initDone : BOOL := FALSE;
    errFull : WORD := 16#8001;
    errEmpty : WORD := 16#8002;
END_VAR

(* Reset error status at start of each cycle *)
error := FALSE;
status := 16#0000;

(* Initialize storage array if not done yet *)
IF NOT initDone THEN
    i := 1;
    WHILE i <= 9 DO
        library[i] := FALSE;
        i := i + 1;
    END_WHILE;
    productNum := 0;
    libFreeNum := 9;
    initDone := TRUE;
END_IF;

(* Handle product storage request *)
IF requestIn AND NOT requestOut THEN
    (* Check if storage is full *)
    IF productNum >= 9 THEN
        error := TRUE;
        status := errFull;
    ELSE
        (* Search for free position from highest to lowest index (FILO) *)
        found := FALSE;
        i := 9;
        WHILE i >= 1 DO
            IF NOT library[i] THEN
                library[i] := TRUE;
                found := TRUE;
                productNum := productNum + 1;
                libFreeNum := libFreeNum - 1;
                EXIT;
            END_IF;
            i := i - 1;
        END_WHILE;

        (* If no free position found despite counter check, set error *)
        IF NOT found THEN
            error := TRUE;
            status := errFull;
        END_IF;
    END_IF;

(* Handle product retrieval request *)
ELSIF requestOut AND NOT requestIn THEN
    (* Check if storage is empty *)
    IF productNum <= 0 THEN
        error := TRUE;
        status := errEmpty;
    ELSE
        (* Search for occupied position from lowest to highest index (FIFO) *)
        found := FALSE;
        i := 1;
        WHILE i <= 9 DO
            IF library[i] THEN
                library[i] := FALSE;
                found := TRUE;
                productNum := productNum - 1;
                libFreeNum := libFreeNum + 1;
                EXIT;
            END_IF;
            i := i + 1;
        END_WHILE;

        (* If no occupied position found despite counter check, set error *)
        IF NOT found THEN
            error := TRUE;
            status := errEmpty;
        END_IF;
    END_IF;

(* Handle concurrent requests - treat as error *)
ELSIF requestIn AND requestOut THEN
    error := TRUE;
    status := 16#8003; (* Concurrent request error *)
END_IF;

(* Validate counters consistency *)
IF (productNum + libFreeNum) <> 9 THEN
    error := TRUE;
    status := 16#8004; (* Counter inconsistency error *)
END_IF;

END_FUNCTION_BLOCK

(* ---- hf_18.st ---- *)
FUNCTION_BLOCK FB_ColorLightControl
VAR_INPUT
    controlButton : BOOL; // Push button for sequence control
END_VAR

VAR_OUTPUT
    greenLight : BOOL; // Green light control signal
    redLight : BOOL; // Red light control signal
    yellowLight : BOOL; // Yellow light control signal
END_VAR

VAR
    state : INT := 1; // State machine control variable
    lastControlButton : BOOL := FALSE; // Previous button state
END_VAR

// Main logic
IF controlButton AND NOT lastControlButton THEN
    // Rising edge detected - execute state transition
    CASE state OF
        1: // State 1: Green Only
            greenLight := TRUE;
            redLight := FALSE;
            yellowLight := FALSE;
            state := 2;

        2: // State 2: Red Only
            greenLight := FALSE;
            redLight := TRUE;
            yellowLight := FALSE;
            state := 3;

        3: // State 3: Yellow Only
            greenLight := FALSE;
            redLight := FALSE;
            yellowLight := TRUE;
            state := 4;

        4: // State 4: All Lights On
            greenLight := TRUE;
            redLight := TRUE;
            yellowLight := TRUE;
            state := 5;

        5: // State 5: All Lights Off
            greenLight := FALSE;
            redLight := FALSE;
            yellowLight := FALSE;
            state := 1;
    END_CASE;
ELSE
    // No rising edge - maintain current light states
    CASE state OF
        1:
            greenLight := TRUE;
            redLight := FALSE;
            yellowLight := FALSE;

        2:
            greenLight := FALSE;
            redLight := TRUE;
            yellowLight := FALSE;

        3:
            greenLight := FALSE;
            redLight := FALSE;
            yellowLight := TRUE;

        4:
            greenLight := TRUE;
            redLight := TRUE;
            yellowLight := TRUE;

        5:
            greenLight := FALSE;
            redLight := FALSE;
            yellowLight := FALSE;
    END_CASE;
END_IF;

// Update last button state for next cycle
lastControlButton := controlButton;

END_FUNCTION_BLOCK

(* ---- hf_19.st ---- *)
FUNCTION_BLOCK FB_DatabaseManager
VAR_INPUT
    dataInput : ARRAY[0..5] OF BYTE;
    storeTrigger : BOOL;
    resetTrigger : BOOL;
END_VAR
VAR_OUTPUT
    usedSpace : INT := 0;
    remainingSpace : INT := 20;
    error : BOOL;
    status : WORD;
END_VAR
VAR_IN_OUT
    dataBase : ARRAY[1..20] OF BYTE;
END_VAR
VAR
    i : INT;
    dataLength : INT;
END_VAR

// Main execution logic
IF resetTrigger THEN
    // Reset operation
    FOR i := 1 TO 20 DO
        dataBase[i] := 0;
    END_FOR;
    usedSpace := 0;
    remainingSpace := 20;
    error := FALSE;
    status := 0;
ELSIF storeTrigger THEN
    // Data storage operation
    dataLength := dataInput[0];

    // Length validation
    IF (dataLength <= 0) OR (dataLength > 5) THEN
        error := TRUE;
        status := 16#8001;
    ELSE
        // Space verification
        IF (usedSpace + dataLength) > 20 THEN
            error := TRUE;
            status := 16#8002;
        ELSE
            // Data storage
            FOR i := 1 TO dataLength DO
                dataBase[usedSpace + i] := dataInput[i];
            END_FOR;

            // Update counters and status
            usedSpace := usedSpace + dataLength;
            remainingSpace := 20 - usedSpace;
            error := FALSE;
            status := 0;
        END_IF;
    END_IF;
END_IF;

END_FUNCTION_BLOCK

(* ---- hf_2.st ---- *)
FUNCTION_BLOCK FindMinMaxValues
VAR_INPUT
    values : ARRAY[1..10] OF DINT;
END_VAR
VAR_OUTPUT
    minValue : DINT;
    minValueIndex : DINT;
    maxValue : DINT;
    maxValueIndex : DINT;
END_VAR
VAR
    i : INT;
END_VAR

BEGIN
    // Initialize with first element
    minValue := values[1];
    minValueIndex := 1;
    maxValue := values[1];
    maxValueIndex := 1;

    // Iterate through remaining elements
    FOR i := 2 TO 10 DO
        // Check for new minimum
        IF values[i] < minValue THEN
            minValue := values[i];
            minValueIndex := i;
        END_IF;

        // Check for new maximum
        IF values[i] > maxValue THEN
            maxValue := values[i];
            maxValueIndex := i;
        END_IF;
    END_FOR;
END_FUNCTION_BLOCK

(* ---- hf_20.st ---- *)
FUNCTION_BLOCK FB_ProductionLineControl
VAR_INPUT
    Mode : BOOL;            // Manual/Auto mode selection
    ForwardButton : BOOL;   // Forward rotation button
    ReverseButton : BOOL;   // Reverse rotation button
    SensorA : BOOL;         // Sensor A input
    SensorB : BOOL;         // Sensor B input
    SensorC : BOOL;         // Sensor C input
    ButtonA : BOOL;         // Button A input
    ButtonB : BOOL;         // Button B input
    ButtonC : BOOL;         // Button C input
END_VAR

VAR_OUTPUT
    MotorForward : BOOL;    // Motor forward output
    MotorReverse : BOOL;    // Motor reverse output
    CompletionLight : BOOL; // Process completion indicator
END_VAR

VAR
    State : INT := 0;       // State machine current state
END_VAR

// Main logic
IF State = 0 THEN
    // Initialization state
    MotorForward := FALSE;
    MotorReverse := FALSE;
    CompletionLight := FALSE;
    State := 1;
END_IF;

IF NOT Mode THEN
    // Manual Mode Operation
    IF ForwardButton AND NOT ReverseButton THEN
        // Forward Motion
        MotorForward := TRUE;
        MotorReverse := FALSE;
    ELSIF ReverseButton AND NOT ForwardButton THEN
        // Reverse Motion
        MotorForward := FALSE;
        MotorReverse := TRUE;
    ELSE
        // Stop Condition (both pressed or neither pressed)
        MotorForward := FALSE;
        MotorReverse := FALSE;
    END_IF;

    // Reset state to 1 when switching to manual mode
    State := 1;
    CompletionLight := FALSE;
ELSE
    // Automatic Mode Operation
    CASE State OF
        1: // Waiting at Station A
            MotorForward := FALSE;
            MotorReverse := FALSE;
            IF SensorA THEN
                State := 2;
            END_IF;

        2: // Processing at Station A
            MotorForward := FALSE;
            MotorReverse := FALSE;
            IF ButtonA THEN
                MotorForward := TRUE;
                MotorReverse := FALSE;
                State := 3;
            END_IF;

        3: // Moving to Station B
            // Keep MotorForward TRUE from previous state
            MotorReverse := FALSE;
            IF SensorB THEN
                MotorForward := FALSE;
                State := 4;
            END_IF;

        4: // Processing at Station B
            MotorForward := FALSE;
            MotorReverse := FALSE;
            IF ButtonB THEN
                MotorForward := TRUE;
                MotorReverse := FALSE;
                State := 5;
            END_IF;

        5: // Moving to Station C
            // Keep MotorForward TRUE from previous state
            MotorReverse := FALSE;
            IF SensorC THEN
                MotorForward := FALSE;
                State := 6;
            END_IF;

        6: // Processing at Station C
            MotorForward := FALSE;
            MotorReverse := FALSE;
            IF ButtonC THEN
                CompletionLight := TRUE;
                State := 7;
            END_IF;

        7: // Cycle Completion
            MotorForward := FALSE;
            MotorReverse := FALSE;
            IF NOT SensorC THEN
                CompletionLight := FALSE;
                State := 1;
            END_IF;
    END_CASE;
END_IF;

END_FUNCTION_BLOCK

(* ---- hf_21.st ---- *)
FUNCTION_BLOCK FB_SplitNumber
VAR_INPUT
    InputNumber : INT;
END_VAR

VAR_OUTPUT
    Thousands : INT;
    Hundreds : INT;
    Tens : INT;
    Ones : INT;
    Min : INT;
    error : BOOL;
    status : WORD;
END_VAR

VAR
    tempNumber : INT;
    minValue : INT;
    digit1 : INT;
    digit2 : INT;
    digit3 : INT;
    digit4 : INT;
END_VAR

// Input validation
IF (InputNumber < 0) OR (InputNumber > 9999) THEN
    // Error condition
    error := TRUE;
    status := 16#8001;
    Thousands := 0;
    Hundreds := 0;
    Tens := 0;
    Ones := 0;
    Min := 0;
ELSE
    // Valid input
    error := FALSE;
    status := 16#0000;

    // Digit separation
    Thousands := InputNumber / 1000;
    tempNumber := InputNumber MOD 1000;
    Hundreds := tempNumber / 100;
    tempNumber := tempNumber MOD 100;
    Tens := tempNumber / 10;
    Ones := tempNumber MOD 10;

    // Minimum non-zero digit detection
    minValue := 32767; // Maximum INT value

    // Check Thousands digit
    IF Thousands > 0 THEN
        minValue := minimal(minValue, Thousands);
    END_IF;

    // Check Hundreds digit
    IF Hundreds > 0 THEN
        minValue := minimal(minValue, Hundreds);
    END_IF;

    // Check Tens digit
    IF Tens > 0 THEN
        minValue := minimal(minValue, Tens);
    END_IF;

    // Check Ones digit
    IF Ones > 0 THEN
        minValue := minimal(minValue, Ones);
    END_IF;

    // Set Min output
    IF minValue = 32767 THEN
        // All digits are zero
        Min := 0;
    ELSE
        Min := minValue;
    END_IF;
END_IF;
END_FUNCTION_BLOCK

FUNCTION minimal : INT
VAR_INPUT
    IN1 : INT;
    IN2 : INT;
END_VAR

IF IN1 <= IN2 THEN
    minimal := IN1;
ELSE
    minimal := IN2;
END_IF;
END_FUNCTION

(* ---- hf_3.st ---- *)
FUNCTION_BLOCK MultiPumpCtrl
VAR_INPUT
    mode : BOOL;
    start : BOOL;
    stop : BOOL;
    priorities : ARRAY[1..5] OF INT;
    selections : ARRAY[1..5] OF BOOL;
END_VAR
VAR_OUTPUT
    RunComds : ARRAY[1..5] OF BOOL;
END_VAR
VAR
    i : INT;
    j : INT;
    maxPriority : INT;
    maxIndex : INT;
    runCount : INT;
    usedInAuto : ARRAY[1..5] OF BOOL;
    tempPriority : INT;
    tempIndex : INT;
    sortedPriorities : ARRAY[1..5] OF INT;
    sortedIndices : ARRAY[1..5] OF INT;
END_VAR

// Main logic
IF stop THEN
    // Stop has highest priority - stop all pumps
    FOR i := 1 TO 5 DO
        RunComds[i] := FALSE;
    END_FOR;
ELSE
    // Initialize arrays
    FOR i := 1 TO 5 DO
        RunComds[i] := FALSE;
        usedInAuto[i] := FALSE;
        sortedIndices[i] := i;
        sortedPriorities[i] := priorities[i];
    END_FOR;

    // Simple bubble sort to sort pumps by priority (descending)
    FOR i := 1 TO 4 DO
        FOR j := i + 1 TO 5 DO
            IF sortedPriorities[i] < sortedPriorities[j] THEN
                // Swap priorities
                tempPriority := sortedPriorities[i];
                sortedPriorities[i] := sortedPriorities[j];
                sortedPriorities[j] := tempPriority;

                // Swap indices to track which pump
                tempIndex := sortedIndices[i];
                sortedIndices[i] := sortedIndices[j];
                sortedIndices[j] := tempIndex;
            END_IF;
        END_FOR;
    END_FOR;

    IF start THEN
        IF NOT mode THEN
            // Manual mode: use selections array directly
            FOR i := 1 TO 5 DO
                RunComds[i] := selections[i];
            END_FOR;
        ELSE
            // Automatic mode: run 3 pumps with highest priorities
            runCount := 0;
            FOR i := 1 TO 5 DO
                IF runCount < 3 THEN
                    RunComds[sortedIndices[i]] := TRUE;
                    runCount := runCount + 1;
                ELSE
                    RunComds[sortedIndices[i]] := FALSE;
                END_IF;
            END_FOR;
        END_IF;
    END_IF;
END_IF;

END_FUNCTION_BLOCK

(* ---- hf_4.st ---- *)
FUNCTION_BLOCK FB_CalculateDayOfYear
VAR_INPUT
    Year : INT;
    Month : INT;
    Day : INT;
END_VAR

VAR_OUTPUT
    DayOfYear : INT;
    error : BOOL;
    status : WORD;
END_VAR

VAR_TEMP
    i : INT;
    IsLeapYear : BOOL;
    MaxDayForMonth : INT;
END_VAR

VAR
    DaysInMonth : ARRAY[1..12] OF INT := [31, 28, 31, 30, 31, 30, 31, 31, 30, 31, 30, 31];
END_VAR

(* Initialize outputs *)
DayOfYear := 0;
error := FALSE;
status := 0;

(* Validate Month - highest priority *)
IF (Month < 1) OR (Month > 12) THEN
    error := TRUE;
    status := 16#8002;
    RETURN;
END_IF;

(* Validate Year - lowest priority *)
IF (Year < 1000) OR (Year > 3000) THEN
    error := TRUE;
    status := 16#8001;
    RETURN;
END_IF;

(* Determine leap year *)
IsLeapYear := ((Year MOD 4) = 0) AND ((Year MOD 100) <> 0);
IsLeapYear := IsLeapYear OR ((Year MOD 400) = 0);

(* Determine maximum day for the given month *)
MaxDayForMonth := DaysInMonth[Month];
IF (Month = 2) AND IsLeapYear THEN
    MaxDayForMonth := 29;
END_IF;

(* Validate Day - second priority *)
IF (Day < 1) OR (Day > MaxDayForMonth) THEN
    error := TRUE;
    status := 16#8003;
    RETURN;
END_IF;

(* Calculate Day of Year *)
FOR i := 1 TO (Month - 1) DO
    DayOfYear := DayOfYear + DaysInMonth[i];
END_FOR;

DayOfYear := DayOfYear + Day;

(* Add extra day for leap year if month is after February *)
IF IsLeapYear AND (Month > 2) THEN
    DayOfYear := DayOfYear + 1;
END_IF;

END_FUNCTION_BLOCK

(* ---- hf_5.st ---- *)
FUNCTION_BLOCK SelectSort
VAR_INPUT
    exe : BOOL;
    seq : ARRAY[1..100] OF INT;
END_VAR
VAR_OUTPUT
    error : BOOL;
    status : WORD;
END_VAR
VAR
    i : INT;
    j : INT;
    minIndex : INT;
    temp : INT;
    n : INT := 100;
    seqLocal : ARRAY[1..100] OF INT;
    exePrev : BOOL;
    sortSuccessful : BOOL;
END_VAR

(* Initialize outputs *)
error := TRUE;
status := 16#8A01;
sortSuccessful := TRUE;

(* Execute sorting on rising edge of exe *)
IF exe AND NOT exePrev THEN
    (* Copy input array to local working array *)
    seqLocal := seq;

    (* Selection sort algorithm *)
    FOR i := 1 TO n-1 DO
        minIndex := i;

        FOR j := i+1 TO n DO
            IF seqLocal[j] < seqLocal[minIndex] THEN
                minIndex := j;
            END_IF;
        END_FOR;

        (* Swap elements if needed *)
        IF minIndex <> i THEN
            temp := seqLocal[i];
            seqLocal[i] := seqLocal[minIndex];
            seqLocal[minIndex] := temp;
        END_IF;
    END_FOR;

    (* Verify the array is sorted in ascending order *)
    sortSuccessful := TRUE;
    FOR i := 1 TO n-1 DO
        IF seqLocal[i] > seqLocal[i+1] THEN
            sortSuccessful := FALSE;
            EXIT;
        END_IF;
    END_FOR;

    (* Update outputs based on sorting result *)
    IF sortSuccessful THEN
        (* Copy sorted array back to output *)
        seq := seqLocal;
        error := FALSE;
        status := 16#0000;
    ELSE
        (* Sorting verification failed *)
        error := TRUE;
        status := 16#8A01;
    END_IF;
END_IF;

(* Store previous execution state *)
exePrev := exe;

END_FUNCTION_BLOCK

(* ---- hf_6.st ---- *)
FUNCTION_BLOCK RandomNumberGenerator
VAR_INPUT
    minValue : DINT;
    maxValue : DINT;
    randomSeed_in : DINT;
END_VAR
VAR_OUTPUT
    error : BOOL;
    status : WORD;
    randomNumber : DINT;
END_VAR
VAR
    internalSeed : DINT;
END_VAR

(* Check for invalid range *)
IF minValue > maxValue THEN
    error := TRUE;
    status := 16#8200;
    randomNumber := 0;
ELSE
    (* Initialize with external seed *)
    internalSeed := randomSeed_in;

    (* Ensure seed is positive *)
    IF internalSeed < 0 THEN
        internalSeed := -internalSeed;
    END_IF;

    (* Simple linear congruential generator algorithm *)
    internalSeed := internalSeed * 1103515245 + 12345;

    (* Generate random number within specified range *)
    randomNumber := minValue + (internalSeed MOD (maxValue - minValue + 1));

    (* Set success status *)
    error := FALSE;
    status := 16#0000;
END_IF;

(* ---- hf_7.st ---- *)
FUNCTION_BLOCK AnalogBatchConverter
VAR_INPUT
    count : INT;
    analogValues : ARRAY[1..10] OF REAL;
END_VAR
VAR_OUTPUT
    channel_enable : ARRAY[1..10] OF BOOL;
    channel_hiLIM : ARRAY[1..10] OF REAL;
    channel_loLIM : ARRAY[1..10] OF REAL;
    channel_bipolar : ARRAY[1..10] OF BOOL;
    channel_measuringMode : ARRAY[1..10] OF INT;
    channel_retVal : ARRAY[1..10] OF WORD;
    channel_outputValue : ARRAY[1..10] OF REAL;
END_VAR
VAR
    i : INT;
    rawValue : REAL;
    scaleFactor : REAL;
END_VAR

FOR i := 1 TO 10 DO
    channel_retVal[i] := 16#0000;
    channel_outputValue[i] := 0.0;

    IF (i <= count) AND channel_enable[i] THEN
        rawValue := analogValues[i];

        CASE channel_measuringMode[i] OF
            0:  // Non-temperature measurement
                IF channel_hiLIM[i] <= channel_loLIM[i] THEN
                    channel_retVal[i] := 16#8002;
                ELSE
                    IF channel_bipolar[i] THEN
                        // Bipolar: map from -27648.0 to 27648.0
                        scaleFactor := (rawValue + 27648.0) / (2.0 * 27648.0);
                    ELSE
                        // Unipolar: map from 0.0 to 27648.0
                        scaleFactor := rawValue / 27648.0;
                    END_IF
                    channel_outputValue[i] := channel_loLIM[i] + scaleFactor * (channel_hiLIM[i] - channel_loLIM[i]);
                END_IF

            1:  // Standard temperature measurement
                channel_outputValue[i] := rawValue / 10.0;

            2:  // Climatic temperature measurement
                channel_outputValue[i] := rawValue / 100.0;

            ELSE
                channel_retVal[i] := 16#8001;
        END_CASE
    END_IF
END_FOR
END_FUNCTION_BLOCK

(* ---- hf_8.st ---- *)
FUNCTION_BLOCK FB_HexDigitAnalyzer
VAR_INPUT
    InputNumber: INT;
END_VAR

VAR_OUTPUT
    Thousands: INT;
    Hundreds: INT;
    Tens: INT;
    Ones: INT;
    MinDigit: INT;
    error: BOOL;
    status: WORD;
END_VAR

VAR
    tempMinValue: INT;
    tempDigit: INT;
END_VAR

METHOD AnalyzeDigits: BOOL
VAR_INPUT
END_VAR
VAR
END_VAR

    // Input validation
    IF (InputNumber < 0) OR (InputNumber > 9999) THEN
        // Error condition
        error := TRUE;
        status := 16#8001;

        // Reset all outputs
        Thousands := 0;
        Hundreds := 0;
        Tens := 0;
        Ones := 0;
        MinDigit := 0;

        RETURN FALSE;
    ELSE
        // Valid input
        error := FALSE;
        status := 16#0000;

        // Digit separation
        Thousands := InputNumber / 1000;
        Hundreds := (InputNumber MOD 1000) / 100;
        Tens := (InputNumber MOD 100) / 10;
        Ones := InputNumber MOD 10;

        // Minimum non-zero digit detection
        tempMinValue := 32767; // Maximum INT value

        // Check thousands digit
        IF Thousands > 0 THEN
            IF Thousands < tempMinValue THEN
                tempMinValue := Thousands;
            END_IF;
        END_IF;

        // Check hundreds digit
        IF Hundreds > 0 THEN
            IF Hundreds < tempMinValue THEN
                tempMinValue := Hundreds;
            END_IF;
        END_IF;

        // Check tens digit
        IF Tens > 0 THEN
            IF Tens < tempMinValue THEN
                tempMinValue := Tens;
            END_IF;
        END_IF;

        // Check ones digit
        IF Ones > 0 THEN
            IF Ones < tempMinValue THEN
                tempMinValue := Ones;
            END_IF;
        END_IF;

        // Set MinDigit output
        IF tempMinValue = 32767 THEN
            // All digits are zero
            MinDigit := 0;
        ELSE
            MinDigit := tempMinValue;
        END_IF;

        RETURN TRUE;
    END_IF;
END_METHOD

// Main execution
AnalyzeDigits();

END_FUNCTION_BLOCK

(* ---- hf_9.st ---- *)
FUNCTION_BLOCK ShellSortFB
VAR_INPUT
    sortDirection : BOOL; (* FALSE = Ascending, TRUE = Descending *)
    arr : ARRAY[1..1000] OF DINT;
END_VAR
VAR_OUTPUT
    error : BOOL;
    status : WORD;
    sorted_arr : ARRAY[1..1000] OF DINT;
END_VAR
VAR
    i : DINT;
    j : DINT;
    gap : DINT;
    temp : DINT;
    n : DINT;
    ascending : BOOL;
    compareCondition : BOOL;
END_VAR

(* Initialize outputs *)
error := FALSE;
status := 16#0000;
sorted_arr := arr;
n := 1000;

(* Fixed size validation - N is fixed at 1000 *)
IF n <= 1 THEN
    error := TRUE;
    status := 16#8200;
    RETURN;
ELSIF n > 1000 THEN
    error := TRUE;
    status := 16#8201;
    RETURN;
END_IF;

(* Determine sort order: FALSE = Ascending, TRUE = Descending *)
ascending := NOT sortDirection;

(* Shell Sort Algorithm *)
gap := n / 2;
WHILE gap > 0 DO
    i := gap + 1;
    WHILE i <= n DO
        temp := sorted_arr[i];
        j := i;

        (* Determine comparison condition based on sort direction *)
        IF ascending THEN
            compareCondition := (j > gap) AND (sorted_arr[j - gap] > temp);
        ELSE
            compareCondition := (j > gap) AND (sorted_arr[j - gap] < temp);
        END_IF;

        WHILE compareCondition DO
            sorted_arr[j] := sorted_arr[j - gap];
            j := j - gap;

            (* Update comparison condition for next iteration *)
            IF ascending THEN
                compareCondition := (j > gap) AND (sorted_arr[j - gap] > temp);
            ELSE
                compareCondition := (j > gap) AND (sorted_arr[j - gap] < temp);
            END_IF;
        END_WHILE;

        sorted_arr[j] := temp;
        i := i + 1;
    END_WHILE;
    gap := gap / 2;
END_WHILE;
END_FUNCTION_BLOCK

(* ---- med_22.st ---- *)
FUNCTION_BLOCK CottonCandyMachine
VAR_INPUT
    SugarLevel : REAL; (* Input for sugar level *)
    SpinningSpeed : INT; (* Input for spinning speed *)
END_VAR
VAR_OUTPUT
    SugarFeeder : BOOL; (* Output to control sugar feeding *)
    MotorSpeed : INT; (* Output to control spinning motor speed *)
END_VAR

(* Main Logic *)
SugarFeeder := SugarLevel < 10.0;

IF SpinningSpeed > 0 THEN
    MotorSpeed := SpinningSpeed;
ELSE
    MotorSpeed := 0;
END_IF;

END_FUNCTION_BLOCK

(* ---- med_23.st ---- *)
FUNCTION_BLOCK SmartIrrigationSystem
VAR_INPUT
    SoilMoistureSensor1 : REAL;
    SoilMoistureSensor2 : REAL;
    WeatherForecast : INT; (* 0: Sunny, 1: Rainy, 2: Cloudy *)
END_VAR

VAR_OUTPUT
    WaterPump : BOOL;
END_VAR

VAR
    SoilMoistureThreshold : REAL := 30.0;
END_VAR

(* Main irrigation logic *)
IF WeatherForecast = 1 THEN
    (* Deactivate pump if rain is forecast *)
    WaterPump := FALSE;
ELSIF WeatherForecast = 0 THEN
    (* Activate pump only if sunny AND at least one sensor below threshold *)
    WaterPump := (SoilMoistureSensor1 < SoilMoistureThreshold) OR
                 (SoilMoistureSensor2 < SoilMoistureThreshold);
ELSE
    (* Keep pump off for cloudy or any other weather condition *)
    WaterPump := FALSE;
END_IF;

END_FUNCTION_BLOCK

(* ---- med_24.st ---- *)
FUNCTION_BLOCK AutomaticDoorControl
VAR_INPUT
    ProximitySensor : BOOL;
    ElapsedTime : DINT; (* milliseconds since door was last opened *)
END_VAR

VAR_OUTPUT
    DoorOpen : BOOL;
END_VAR

VAR
    DoorOpenDuration : DINT := 5000; (* 5 seconds in milliseconds *)
    eState : (stDoorClosed, stDoorOpen, stDoorClosing);
END_VAR

(* Main state machine logic *)
CASE eState OF
    stDoorClosed:
        DoorOpen := FALSE;
        IF ProximitySensor THEN
            eState := stDoorOpen;
        END_IF;

    stDoorOpen:
        DoorOpen := TRUE;
        IF NOT ProximitySensor AND (ElapsedTime >= DoorOpenDuration) THEN
            eState := stDoorClosing;
        END_IF;

    stDoorClosing:
        DoorOpen := FALSE;
        IF NOT ProximitySensor THEN
            eState := stDoorClosed;
        ELSIF ProximitySensor THEN
            eState := stDoorOpen;
        END_IF;
END_CASE;

END_FUNCTION_BLOCK

(* ---- med_25.st ---- *)
FUNCTION_BLOCK WastewaterControl
VAR_INPUT
    InFlow : REAL;
    OutFlow : REAL;
    pH : REAL;
    TankLvl : REAL;
END_VAR

VAR_OUTPUT
    Pump1 : BOOL;
    Pump2 : BOOL;
    Valve1 : BOOL;
    Valve2 : BOOL;
END_VAR

VAR
    LowInFlow : REAL := 100.0;
    HighOutFlow : REAL := 90.0;
    DesiredPH : REAL := 7.0;
    HighTankLvl : REAL := 80.0;
END_VAR

// Main control logic
Pump1 := InFlow < LowInFlow;
Pump2 := OutFlow > HighOutFlow;
Valve1 := pH < DesiredPH;
Valve2 := TankLvl > HighTankLvl;

END_FUNCTION_BLOCK

(* ---- med_26.st ---- *)
FUNCTION_BLOCK BookSorting
VAR_INPUT
    RFID1 : BOOL;
    RFID2 : BOOL;
    RFID3 : BOOL;
END_VAR

VAR_OUTPUT
    Motor : BOOL;
    Bin1 : BOOL;
    Bin2 : BOOL;
    Bin3 : BOOL;
END_VAR

VAR
    anyRFID : BOOL;
END_VAR

    // Determine if any RFID reader is active
    anyRFID := RFID1 OR RFID2 OR RFID3;

    // Control conveyor motor based on RFID detection
    Motor := anyRFID;

    // Control sorting bins with priority logic (only one bin open at a time)
    IF RFID1 THEN
        Bin1 := TRUE;
        Bin2 := FALSE;
        Bin3 := FALSE;
    ELSIF RFID2 THEN
        Bin1 := FALSE;
        Bin2 := TRUE;
        Bin3 := FALSE;
    ELSIF RFID3 THEN
        Bin1 := FALSE;
        Bin2 := FALSE;
        Bin3 := TRUE;
    ELSE
        // No RFID detection - close all bins
        Bin1 := FALSE;
        Bin2 := FALSE;
        Bin3 := FALSE;
    END_IF;

END_FUNCTION_BLOCK

(* ---- med_27.st ---- *)
FUNCTION_BLOCK FlowerArrangingMachine
VAR_INPUT
    FlowerTypeSensor : INT; (* Input for detecting flower type *)
    FlowerColorSensor : INT; (* Input for detecting flower color *)
END_VAR
VAR_OUTPUT
    ArrangingMechanism : INT; (* Output for controlling arranging mechanism *)
    ConveyorBelt : BOOL; (* Output for controlling conveyor belt *)
END_VAR

VAR
    tempArrangingMechanism : INT;
END_VAR

(* Determine ArrangingMechanism value based on sensor inputs *)
IF (FlowerTypeSensor = 1) AND (FlowerColorSensor = 1) THEN
    tempArrangingMechanism := 1;
ELSIF (FlowerTypeSensor = 1) AND (FlowerColorSensor = 2) THEN
    tempArrangingMechanism := 2;
ELSIF (FlowerTypeSensor = 2) AND (FlowerColorSensor = 1) THEN
    tempArrangingMechanism := 3;
ELSIF (FlowerTypeSensor = 2) AND (FlowerColorSensor = 2) THEN
    tempArrangingMechanism := 4;
ELSE
    tempArrangingMechanism := 0;
END_IF;

(* Assign the calculated value to the output *)
ArrangingMechanism := tempArrangingMechanism;

(* Control ConveyorBelt based on ArrangingMechanism *)
ConveyorBelt := (ArrangingMechanism <> 0);

END_FUNCTION_BLOCK

(* ---- med_28.st ---- *)
FUNCTION_BLOCK HomeBrewingSystem
VAR_INPUT
    TemperatureSensor : REAL; (* Input for temperature measurement *)
    WaterFlowSensor : REAL; (* Input for water flow measurement *)
    BrewingStartTime : TIME; (* Input for brewing start time *)
    BrewingDuration : TIME; (* Input for brewing duration *)
END_VAR
VAR_OUTPUT
    HeatingElement : BOOL; (* Output for heating element *)
    AgitationMotor : BOOL; (* Output for agitation motor *)
    HopsDispenser : BOOL; (* Output for hops dispenser *)
    FermentationTank : BOOL; (* Output for fermentation tank *)
END_VAR
VAR
    CurrentTime : TIME;
    ElapsedBrewingTime : TIME;
END_VAR

(* Calculate elapsed brewing time *)
CurrentTime := TIME(); (* Get current PLC time *)
IF BrewingStartTime <= CurrentTime THEN
    ElapsedBrewingTime := CurrentTime - BrewingStartTime;
ELSE
    ElapsedBrewingTime := T#0s; (* Handle invalid start time *)
END_IF

(* Control Heating Element based on temperature *)
IF TemperatureSensor < 65.0 THEN
    HeatingElement := TRUE;
ELSE
    HeatingElement := FALSE;
END_IF;

(* Control Agitation Motor based on water flow *)
IF WaterFlowSensor > 0.5 THEN
    AgitationMotor := TRUE;
ELSE
    AgitationMotor := FALSE;
END_IF;

(* Control Hops Dispenser after 5 hours of brewing *)
IF (ElapsedBrewingTime >= T#5h) AND (ElapsedBrewingTime <= BrewingDuration) THEN
    HopsDispenser := TRUE;
ELSE
    HopsDispenser := FALSE;
END_IF;

(* Control Fermentation Tank after 48 hours of brewing *)
IF (ElapsedBrewingTime >= T#48h) AND (ElapsedBrewingTime <= BrewingDuration) THEN
    FermentationTank := TRUE;
ELSE
    FermentationTank := FALSE;
END_IF;

END_FUNCTION_BLOCK

(* ---- med_29.st ---- *)
FUNCTION_BLOCK DocumentFilingSystem
VAR_INPUT
    DocumentInlet : BOOL; (* Input to detect the arrival of a document *)
    CategorySelector : INT; (* Input to select the document category *)
END_VAR
VAR_OUTPUT
    ConveyorMotor : BOOL; (* Output to control the conveyor motor *)
    StorageBin1 : BOOL; (* Output to activate storage bin 1 *)
    StorageBin2 : BOOL; (* Output to activate storage bin 2 *)
    StorageBin3 : BOOL; (* Output to activate storage bin 3 *)
    StorageBin4 : BOOL; (* Output to activate storage bin 4 *)
END_VAR
VAR
    CategoryValid : BOOL; (* Internal variable to validate category *)
END_VAR

(* Validate category selector *)
CategoryValid := (CategorySelector >= 1) AND (CategorySelector <= 4);

(* Main control logic *)
IF DocumentInlet AND CategoryValid THEN
    ConveyorMotor := TRUE;

    (* Activate appropriate storage bin based on category *)
    CASE CategorySelector OF
        1:
            StorageBin1 := TRUE;
            StorageBin2 := FALSE;
            StorageBin3 := FALSE;
            StorageBin4 := FALSE;
        2:
            StorageBin1 := FALSE;
            StorageBin2 := TRUE;
            StorageBin3 := FALSE;
            StorageBin4 := FALSE;
        3:
            StorageBin1 := FALSE;
            StorageBin2 := FALSE;
            StorageBin3 := TRUE;
            StorageBin4 := FALSE;
        4:
            StorageBin1 := FALSE;
            StorageBin2 := FALSE;
            StorageBin3 := FALSE;
            StorageBin4 := TRUE;
        ELSE
            (* Fallback for any unexpected value *)
            StorageBin1 := FALSE;
            StorageBin2 := FALSE;
            StorageBin3 := FALSE;
            StorageBin4 := FALSE;
    END_CASE;
ELSE
    (* Deactivate all outputs when no document or invalid category *)
    ConveyorMotor := FALSE;
    StorageBin1 := FALSE;
    StorageBin2 := FALSE;
    StorageBin3 := FALSE;
    StorageBin4 := FALSE;
END_IF;

END_FUNCTION_BLOCK

(* ---- med_30.st ---- *)
FUNCTION_BLOCK MuseumClimateControl
VAR_INPUT
    HumiditySensor : REAL;
    TemperatureSensor : REAL;
    LightSensor : BOOL;
END_VAR

VAR_OUTPUT
    HVACSystem : BOOL;
    Humidifier : BOOL;
    Dehumidifier : BOOL;
    LightControl : BOOL;
END_VAR

VAR
    TargetHumidity : REAL := 50.0;
    TargetTemperature : REAL := 20.0;
    LightThreshold : BOOL := TRUE;
END_VAR

// Humidity control logic
IF HumiditySensor < TargetHumidity THEN
    Humidifier := TRUE;
    Dehumidifier := FALSE;
ELSIF HumiditySensor > TargetHumidity THEN
    Humidifier := FALSE;
    Dehumidifier := TRUE;
ELSE
    Humidifier := FALSE;
    Dehumidifier := FALSE;
END_IF;

// Temperature control logic
IF TemperatureSensor <> TargetTemperature THEN
    HVACSystem := TRUE;
ELSE
    HVACSystem := FALSE;
END_IF;

// Lighting control logic
IF LightSensor AND LightThreshold THEN
    LightControl := FALSE;
ELSE
    LightControl := TRUE;
END_IF;

END_FUNCTION_BLOCK

(* ---- med_31.st ---- *)
FUNCTION_BLOCK ChargingStationControl
VAR_INPUT
    EVConnected : BOOL;
    EVVoltage : REAL;
    EVCurrent : REAL;
    EVStateOfCharge : REAL;
    ChargingTimer : TIME;
END_VAR

VAR_OUTPUT
    EVCharging : BOOL;
END_VAR

VAR
    VoltageOK : BOOL;
    CurrentOK : BOOL;
    SOCNotFull : BOOL;
    TimerOK : BOOL;
END_VAR

(* Evaluate individual conditions *)
VoltageOK := EVVoltage > 350.0;
CurrentOK := EVCurrent <= 32.0;
SOCNotFull := EVStateOfCharge < 100.0;
TimerOK := ChargingTimer <= T#2h;

(* Main charging control logic *)
IF EVConnected AND VoltageOK AND CurrentOK AND SOCNotFull AND TimerOK THEN
    EVCharging := TRUE;
ELSE
    EVCharging := FALSE;
END_IF;

END_FUNCTION_BLOCK

(* ---- med_32.st ---- *)
FUNCTION_BLOCK GreenhouseWateringSystem
VAR_INPUT
    SoilMoistureSensor : REAL;   (* Input for soil moisture level (0-100%) *)
END_VAR
VAR_OUTPUT
    SprinklersOn : BOOL := FALSE; (* Output for controlling sprinklers - on/off *)
END_VAR
VAR
    ResponseDelay : TIME := T#5s;  (* Example response delay for the system *)
    LastMoistureReading : REAL;
    tDelay : TON;
    bDelayActive : BOOL := FALSE;
    eState : (eIdle, eActivating, eActive, eDeactivating) := eIdle;
END_VAR

(* Timer initialization *)
tDelay(IN:=bDelayActive, PT:=ResponseDelay);

(* Main state machine logic *)
CASE eState OF
    eIdle:
        SprinklersOn := FALSE;
        bDelayActive := FALSE;
        LastMoistureReading := SoilMoistureSensor;

        IF SoilMoistureSensor < 30.0 THEN
            eState := eActivating;
            bDelayActive := TRUE;
        ELSIF SoilMoistureSensor > 70.0 THEN
            eState := eIdle; (* Already in idle, but kept for clarity *)
        END_IF;

    eActivating:
        SprinklersOn := FALSE;
        LastMoistureReading := SoilMoistureSensor;

        IF tDelay.Q THEN
            eState := eActive;
            bDelayActive := FALSE;
        END_IF;

        IF SoilMoistureSensor > 70.0 THEN
            eState := eIdle;
            bDelayActive := FALSE;
        END_IF;

    eActive:
        SprinklersOn := TRUE;
        bDelayActive := FALSE;
        LastMoistureReading := SoilMoistureSensor;

        IF SoilMoistureSensor > 70.0 THEN
            eState := eDeactivating;
            bDelayActive := TRUE;
        END_IF;

    eDeactivating:
        SprinklersOn := TRUE;
        LastMoistureReading := SoilMoistureSensor;

        IF tDelay.Q THEN
            eState := eIdle;
            bDelayActive := FALSE;
        END_IF;

        IF SoilMoistureSensor < 30.0 THEN
            eState := eActive;
            bDelayActive := FALSE;
        END_IF;

END_CASE;
END_FUNCTION_BLOCK

(* ---- med_33.st ---- *)
FUNCTION_BLOCK RoboticArmColorSorting
VAR_INPUT
    ColorSensorRed : BOOL;   (* Input: Red color sensor *)
    ColorSensorGreen : BOOL;  (* Input: Green color sensor *)
    ColorSensorBlue : BOOL;   (* Input: Blue color sensor *)
END_VAR

VAR_OUTPUT
    RoboticArmMove : BOOL := FALSE;     (* Output: Control for robotic arm movement *)
    BinRed : BOOL := FALSE;           (* Output: Activate red bin *)
    BinGreen : BOOL := FALSE;         (* Output: Activate green bin *)
    BinBlue : BOOL := FALSE;          (* Output: Activate blue bin *)
END_VAR

VAR
    AnyColorDetected : BOOL;
END_VAR

(* Main Logic *)
AnyColorDetected := ColorSensorRed OR ColorSensorGreen OR ColorSensorBlue;

RoboticArmMove := AnyColorDetected;

(* Activate bins based on exclusive color detection *)
BinRed := ColorSensorRed AND NOT ColorSensorGreen AND NOT ColorSensorBlue;
BinGreen := ColorSensorGreen AND NOT ColorSensorRed AND NOT ColorSensorBlue;
BinBlue := ColorSensorBlue AND NOT ColorSensorRed AND NOT ColorSensorGreen;

END_FUNCTION_BLOCK

(* ---- med_34.st ---- *)
FUNCTION_BLOCK CoffeeMachineControl
VAR_INPUT
    StartButton : BOOL;
    ElapsedTime : DINT; (* Time elapsed since the start of the current process, in milliseconds *)
END_VAR

VAR_OUTPUT
    WaterHeating : BOOL;
    GrinderRunning : BOOL;
    Brewing : BOOL;
    WaterHeated : BOOL;
    GrinderFinished : BOOL;
    CoffeeReady : BOOL;
END_VAR

VAR
    WaterHeatingDuration : DINT := 30000; (* 30 seconds in milliseconds *)
    GrinderDuration : DINT := 15000; (* 15 seconds in milliseconds *)
    BrewingDuration : DINT := 60000; (* 60 seconds in milliseconds *)
    CurrentState : INT := 0;
    ProcessStartTime : DINT := 0;
END_VAR

(* Reset all outputs when start button is not pressed *)
IF NOT StartButton THEN
    CurrentState := 0;
    ProcessStartTime := 0;
    WaterHeating := FALSE;
    GrinderRunning := FALSE;
    Brewing := FALSE;
    WaterHeated := FALSE;
    GrinderFinished := FALSE;
    CoffeeReady := FALSE;
ELSE
    CASE CurrentState OF
        0: (* Idle - waiting for start *)
            WaterHeating := FALSE;
            GrinderRunning := FALSE;
            Brewing := FALSE;
            WaterHeated := FALSE;
            GrinderFinished := FALSE;
            CoffeeReady := FALSE;

            IF StartButton THEN
                CurrentState := 1;
                ProcessStartTime := ElapsedTime;
            END_IF;

        1: (* Water Heating State *)
            WaterHeating := TRUE;
            GrinderRunning := FALSE;
            Brewing := FALSE;
            WaterHeated := FALSE;

            IF (ElapsedTime - ProcessStartTime) >= WaterHeatingDuration THEN
                WaterHeating := FALSE;
                WaterHeated := TRUE;
                CurrentState := 2;
                ProcessStartTime := ElapsedTime;
            END_IF;

        2: (* Grinder Running State *)
            WaterHeating := FALSE;
            GrinderRunning := TRUE;
            Brewing := FALSE;
            GrinderFinished := FALSE;

            IF (ElapsedTime - ProcessStartTime) >= GrinderDuration THEN
                GrinderRunning := FALSE;
                GrinderFinished := TRUE;
                CurrentState := 3;
                ProcessStartTime := ElapsedTime;
            END_IF;

        3: (* Brewing State *)
            WaterHeating := FALSE;
            GrinderRunning := FALSE;
            Brewing := TRUE;
            CoffeeReady := FALSE;

            IF (ElapsedTime - ProcessStartTime) >= BrewingDuration THEN
                Brewing := FALSE;
                CoffeeReady := TRUE;
                CurrentState := 0;
                ProcessStartTime := 0;
            END_IF;
    END_CASE;
END_IF;

END_FUNCTION_BLOCK

(* ---- med_35.st ---- *)
FUNCTION_BLOCK FB_SimpleCalculation
VAR_INPUT
    INPUT_VAR1 : INT := 2;
    VAR2 : INT := 0;
END_VAR

VAR_OUTPUT
    OUTPUT_VAR1 : INT;
    OUTPUT_VAR2 : INT;
END_VAR

VAR
    COUNTER2 : INT := 0;
    i : INT;
END_VAR

// First calculation: Multiply INPUT_VAR1 by 2 for 5 iterations
OUTPUT_VAR1 := INPUT_VAR1;
FOR i := 1 TO 5 DO
    OUTPUT_VAR1 := OUTPUT_VAR1 * 2;
END_FOR;

// Second calculation: Increment VAR2 by 1 for 5 iterations
OUTPUT_VAR2 := VAR2;
FOR i := 1 TO 5 DO
    OUTPUT_VAR2 := OUTPUT_VAR2 + 1;
END_FOR;
END_FUNCTION_BLOCK

(* ---- med_36.st ---- *)
FUNCTION_BLOCK FB_ExpandedPoint
    VAR_INPUT
        INPUT_VAR2 : INT;
        INPUT_VAR1_X : INT;
        INPUT_VAR1_Y : INT;
        INPUT_VAR3_X : INT := 1;
        INPUT_VAR3_Y : INT := 2;
    END_VAR

    VAR_OUTPUT
        OUTPUT_VAR2 : INT;
        OUTPUT_VAR1_X : INT;
        OUTPUT_VAR1_Y : INT;
        OUTPUT_VAR3_X : INT;
        OUTPUT_VAR3_Y : INT;
    END_VAR

    METHOD Execute : BOOL
        VAR_INPUT
        END_VAR
        VAR_OUTPUT
        END_VAR
        VAR
        END_VAR
        OUTPUT_VAR2 := INPUT_VAR2;
        OUTPUT_VAR1_X := 1;
        OUTPUT_VAR1_Y := 2;
        OUTPUT_VAR3_X := 100;
        OUTPUT_VAR3_Y := -7000;
        Execute := TRUE;
    END_METHOD
END_FUNCTION_BLOCK

(* ---- med_37.st ---- *)
FUNCTION_BLOCK FB_RealValueAdjuster
VAR_INPUT
    x_in : REAL;
END_VAR

VAR_OUTPUT
    x_out : REAL;
END_VAR

VAR
    x_temp : REAL;
    i_temp : INT;
END_VAR

x_temp := x_in;

// First condition: if exactly 0.0, add 1.0
IF x_temp = 0.0 THEN
    x_temp := x_temp + 1.0;
END_IF;

// Second condition: if not 0.0, also add 1.0
IF x_temp <> 0.0 THEN
    x_temp := x_temp + 1.0;
END_IF;

// Convert to integer and check
i_temp := REAL_TO_INT(x_temp);
IF i_temp <> 0 THEN
    x_temp := x_temp + 1.0;
END_IF;

x_out := x_temp;

END_FUNCTION_BLOCK

(* ---- med_38.st ---- *)
FUNCTION_BLOCK SolarPanelTracking
VAR_INPUT
    SolarIntensity : REAL;      (* Input: Solar intensity in percentage *)
    CurrentTime : TIME;         (* Input: Current time of day *)
END_VAR

VAR_OUTPUT
    PanelAngle : REAL := 0.0;   (* Output: Panel angle in degrees *)
END_VAR

VAR
    SunriseTime : TIME := T#6H;    (* Sunrise time set to 6 AM *)
    SunsetTime : TIME := T#18H;    (* Sunset time set to 6 PM *)
    NoonTime : TIME := T#12H;      (* Noon time set to 12 PM *)
    MorningAngle : REAL := 30.0;   (* Angle during morning *)
    NoonAngle : REAL := 60.0;      (* Angle during noon *)
    EveningAngle : REAL := 30.0;   (* Angle during evening *)
END_VAR

(* Main logic *)
IF (CurrentTime < SunriseTime) OR (CurrentTime >= SunsetTime) THEN
    (* Nighttime: set angle to zero *)
    PanelAngle := 0.0;
ELSE
    (* Daytime logic *)
    IF SolarIntensity >= 90.0 THEN
        (* High intensity: use noon angle *)
        PanelAngle := NoonAngle;
    ELSE
        (* Normal intensity: time-based angle selection *)
        IF CurrentTime < NoonTime THEN
            (* Morning: before noon *)
            PanelAngle := MorningAngle;
        ELSE
            (* Evening: after noon *)
            PanelAngle := EveningAngle;
        END_IF;
    END_IF;
END_IF;

(* Ensure angle stays within valid range 0-90 degrees *)
IF PanelAngle < 0.0 THEN
    PanelAngle := 0.0;
ELSIF PanelAngle > 90.0 THEN
    PanelAngle := 90.0;
END_IF;

END_FUNCTION_BLOCK

(* ---- med_39.st ---- *)
FUNCTION_BLOCK WindTurbineControl
VAR_INPUT
    WindSpeedSensor : REAL; (* Input for measuring wind speed *)
    GeneratorSpeedSensor : REAL; (* Input for measuring generator speed *)
END_VAR

VAR_OUTPUT
    BladePitch : INT; (* Output for blade pitch control (degrees) *)
    GeneratorSpeed : REAL; (* Output for generator speed control (RPM) *)
END_VAR

VAR
    (* Internal variables can be added here if needed *)
END_VAR

(* Main control logic *)
IF WindSpeedSensor > 5.0 THEN
    (* High wind speed: > 5.0 m/s *)
    BladePitch := 5;
    GeneratorSpeed := 1000.0;
ELSIF WindSpeedSensor > 3.0 THEN
    (* Moderate wind speed: > 3.0 and <= 5.0 m/s *)
    BladePitch := 0;
    GeneratorSpeed := 800.0;
ELSE
    (* Low wind speed: <= 3.0 m/s *)
    BladePitch := -5;
    GeneratorSpeed := 500.0;
END_IF;

END_FUNCTION_BLOCK

(* ---- med_40.st ---- *)
FUNCTION_BLOCK RockClimbingWallControl
VAR_INPUT
    UserWeightSensor : REAL; (* Input for measuring the user's weight *)
    WallDifficultyLevel : INT; (* Input for setting the wall's initial difficulty level *)
    WallHeight : REAL; (* Input for setting the wall's height *)
    RouteSelector : INT; (* Input for selecting a climbing route *)
END_VAR
VAR_OUTPUT
    ClimbingMotorSpeed : REAL; (* Output for controlling the climbing wall motor speed *)
    WallLights : BOOL; (* Output for controlling wall lighting *)
END_VAR

VAR
    InternalDifficultyLevel : INT;
END_VAR

(* Determine motor speed based on user weight *)
IF UserWeightSensor > 60.0 THEN
    ClimbingMotorSpeed := 1.0;
ELSE
    ClimbingMotorSpeed := 0.8;
END_IF;

(* Determine difficulty level based on selected route *)
CASE RouteSelector OF
    1: InternalDifficultyLevel := 1;
    2: InternalDifficultyLevel := 2;
    3: InternalDifficultyLevel := 3;
    ELSE
        InternalDifficultyLevel := WallDifficultyLevel; (* Fallback to input level *)
END_CASE;

(* Control wall lights based on wall height *)
IF WallHeight > 5.0 THEN
    WallLights := TRUE;
ELSE
    WallLights := FALSE;
END_IF;

END_FUNCTION_BLOCK

(* ---- med_41.st ---- *)
FUNCTION_BLOCK FishTankControl
VAR_INPUT
    OxygenLevel : REAL; (* Input for oxygen level in the tank *)
    WaterTemperature : REAL; (* Input for water temperature *)
    FeedingTime : TIME; (* Time for scheduled feeding *)
    CurrentTime : TIME; (* Current system time *)
END_VAR
VAR_OUTPUT
    OxygenValve : BOOL; (* Output to control oxygen supply *)
    Heater : BOOL; (* Output to control the heater *)
    Feeder : BOOL; (* Output to control the fish feeder *)
END_VAR

// Main logic
IF OxygenLevel < 5.0 THEN
    OxygenValve := TRUE;
ELSE
    OxygenValve := FALSE;
END_IF;

IF WaterTemperature < 25.0 THEN
    Heater := TRUE;
ELSE
    Heater := FALSE;
END_IF;

IF CurrentTime >= FeedingTime THEN
    Feeder := TRUE;
ELSE
    Feeder := FALSE;
END_IF;

END_FUNCTION_BLOCK

(* ---- med_42.st ---- *)
FUNCTION_BLOCK RetractableRoofControl
VAR_INPUT
    RainSensor : BOOL; (* Input to detect rain *)
    WindSensor : BOOL; (* Input to detect wind *)
    TemperatureSensor : REAL; (* Input to measure temperature *)
END_VAR
VAR_OUTPUT
    RoofMotor : BOOL; (* Output to control the roof motor *)
END_VAR

// Main logic implementation
IF RainSensor AND WindSensor THEN
    RoofMotor := FALSE; (* Close completely when raining and windy *)
ELSIF RainSensor AND NOT WindSensor THEN
    RoofMotor := TRUE; (* Partially close when raining but not windy *)
ELSIF NOT RainSensor AND TemperatureSensor < 20.0 THEN
    RoofMotor := TRUE; (* Close slightly when not raining and temperature below 20°C *)
ELSIF NOT RainSensor AND TemperatureSensor >= 20.0 THEN
    RoofMotor := FALSE; (* Fully open when not raining and temperature 20°C or above *)
ELSE
    RoofMotor := FALSE; (* Default safe state *)
END_IF;

END_FUNCTION_BLOCK

(* ---- med_43.st ---- *)
FUNCTION_BLOCK SandwichMaker
VAR_INPUT
    BreadFeeder : BOOL; (* Input: Detects the presence of bread slices *)
    Ingredient1 : BOOL; (* Input: Detects the presence of Ingredient 1 (e.g., cheese) *)
    Ingredient2 : BOOL; (* Input: Detects the presence of Ingredient 2 (e.g., lettuce) *)
    Ingredient3 : BOOL; (* Input: Detects the presence of Ingredient 3 (e.g., tomatoes) *)
    Condiment1 : BOOL; (* Input: Detects the presence of Condiment 1 (e.g., mayo) *)
    Condiment2 : BOOL; (* Input: Detects the presence of Condiment 2 (e.g., mustard) *)
END_VAR
VAR_OUTPUT
    ConveyorMotor : BOOL; (* Output: Controls the conveyor belt motor *)
    AssembleMotor : BOOL; (* Output: Controls the sandwich assembly motor *)
END_VAR
VAR
    SliceCount : INT := 0; (* Counter for bread slices *)
    fbBreadRTrig : R_TRIG; (* Rising edge detector for bread detection *)
END_VAR

(* Detect rising edge of BreadFeeder to count slices *)
fbBreadRTrig(CLK := BreadFeeder);

(* Control conveyor motor based on bread presence *)
ConveyorMotor := BreadFeeder;

(* Increment slice count when bread is newly detected *)
IF fbBreadRTrig.Q THEN
    SliceCount := SliceCount + 1;
END_IF;

(* Control assembly motor based on conditions *)
AssembleMotor := (SliceCount >= 2) AND
                 Ingredient1 AND
                 Ingredient2 AND
                 Ingredient3 AND
                 Condiment1 AND
                 Condiment2;

(* Reset slice count after assembly starts to prepare for next sandwich *)
IF AssembleMotor THEN
    SliceCount := 0;
END_IF;

END_FUNCTION_BLOCK

(* ---- med_44.st ---- *)
FUNCTION_BLOCK DroneChargingStation
VAR_INPUT
    Drone1BatteryLevel : INT := 0; (* Battery level of Drone 1 (0-100%) *)
    Drone2BatteryLevel : INT := 0; (* Battery level of Drone 2 (0-100%) *)
    Drone3BatteryLevel : INT := 0; (* Battery level of Drone 3 (0-100%) *)
    ChargingTime : TIME := T#30s; (* Charging time required for each drone *)
END_VAR
VAR_OUTPUT
    Drone1Status : BOOL := FALSE; (* Status of Drone 1 *)
    Drone2Status : BOOL := FALSE; (* Status of Drone 2 *)
    Drone3Status : BOOL := FALSE; (* Status of Drone 3 *)
    ChargingStationStatus : BOOL := FALSE; (* Charging station status *)
    DroneDeployed : BOOL := FALSE; (* Indicates if a drone is deployed *)
END_VAR
VAR
    TimeRemaining : TIME := T#0s; (* Remaining charging time for the current charging operation *)
    CurrentChargingDrone : INT := 0; (* 0 = none, 1 = Drone1, 2 = Drone2, 3 = Drone3 *)
    InternalDeployed : BOOL := FALSE; (* Internal deployment status *)
END_VAR

(* Check if any deployed drone has critically low battery *)
IF InternalDeployed THEN
    IF (Drone1BatteryLevel < 10) OR (Drone2BatteryLevel < 10) OR (Drone3BatteryLevel < 10) THEN
        InternalDeployed := FALSE;
    END_IF;
END_IF;
DroneDeployed := InternalDeployed;

(* Charging station logic *)
IF NOT ChargingStationStatus THEN
    (* Station is free - check for drones needing charge *)
    IF (Drone1BatteryLevel < 20) AND (CurrentChargingDrone = 0) THEN
        Drone1Status := TRUE;
        ChargingStationStatus := TRUE;
        CurrentChargingDrone := 1;
        TimeRemaining := ChargingTime;
    ELSIF (Drone2BatteryLevel < 20) AND (CurrentChargingDrone = 0) THEN
        Drone2Status := TRUE;
        ChargingStationStatus := TRUE;
        CurrentChargingDrone := 2;
        TimeRemaining := ChargingTime;
    ELSIF (Drone3BatteryLevel < 20) AND (CurrentChargingDrone = 0) THEN
        Drone3Status := TRUE;
        ChargingStationStatus := TRUE;
        CurrentChargingDrone := 3;
        TimeRemaining := ChargingTime;
    END_IF;
ELSE
    (* Station is busy - manage charging timer *)
    IF TimeRemaining > T#0s THEN
        TimeRemaining := TimeRemaining - T#1ms;
    ELSE
        (* Charging complete *)
        Drone1Status := FALSE;
        Drone2Status := FALSE;
        Drone3Status := FALSE;
        ChargingStationStatus := FALSE;
        CurrentChargingDrone := 0;
    END_IF;
END_IF;

(* Deployment logic - can only deploy if station is not charging *)
IF NOT ChargingStationStatus AND NOT InternalDeployed THEN
    (* Check if any drone has sufficient battery for deployment *)
    IF (Drone1BatteryLevel >= 80) OR (Drone2BatteryLevel >= 80) OR (Drone3BatteryLevel >= 80) THEN
        InternalDeployed := TRUE;
    END_IF;
END_IF;

END_FUNCTION_BLOCK

(* ---- med_45.st ---- *)
FUNCTION_BLOCK AutomatedSmoothieMaker
VAR_INPUT
    BananaAvailable : BOOL;
    BerryMixAvailable : BOOL;
    SpinachAvailable : BOOL;
    YogurtAvailable : BOOL;
    CustomerPreference : INT;
END_VAR

VAR_OUTPUT
    BlenderMotor : BOOL;
    Dispenser : BOOL;
END_VAR

VAR
    RecipeValid : BOOL;
    IngredientsAvailable : BOOL;
END_VAR

RecipeValid := FALSE;
IngredientsAvailable := FALSE;

CASE CustomerPreference OF
    1:
        RecipeValid := TRUE;
        IngredientsAvailable := BananaAvailable AND BerryMixAvailable AND YogurtAvailable;
    2:
        RecipeValid := TRUE;
        IngredientsAvailable := BerryMixAvailable AND SpinachAvailable AND YogurtAvailable;
    3:
        RecipeValid := TRUE;
        IngredientsAvailable := BananaAvailable AND SpinachAvailable AND YogurtAvailable;
    ELSE
        RecipeValid := FALSE;
        IngredientsAvailable := FALSE;
END_CASE;

IF RecipeValid AND IngredientsAvailable THEN
    Dispenser := TRUE;
    BlenderMotor := TRUE;
ELSE
    Dispenser := FALSE;
    BlenderMotor := FALSE;
END_IF;

END_FUNCTION_BLOCK

(* ---- med_46.st ---- *)
FUNCTION_BLOCK PrecisionEngravingMachine
VAR_INPUT
    DesignSelection : INT;
END_VAR

VAR_OUTPUT
    ZAxisMotor : BOOL;
    EngravingMotor : BOOL;
    EngravingDepth : REAL;
    EngravingSpeed : REAL;
END_VAR

VAR
    CalculatedDepth : REAL;
    CalculatedSpeed : REAL;
END_VAR

// Main logic for design-based parameter selection and motor control
CASE DesignSelection OF
    1:
        CalculatedSpeed := 10.0;
        CalculatedDepth := 0.1;
        ZAxisMotor := TRUE;
        EngravingMotor := TRUE;
    2:
        CalculatedSpeed := 8.0;
        CalculatedDepth := 0.2;
        ZAxisMotor := TRUE;
        EngravingMotor := TRUE;
    3:
        CalculatedSpeed := 12.0;
        CalculatedDepth := 0.15;
        ZAxisMotor := TRUE;
        EngravingMotor := TRUE;
ELSE
    CalculatedSpeed := 0.0;
    CalculatedDepth := 0.0;
    ZAxisMotor := FALSE;
    EngravingMotor := FALSE;
END_CASE;

// Update output parameters based on calculated values
EngravingSpeed := CalculatedSpeed;
EngravingDepth := CalculatedDepth;

END_FUNCTION_BLOCK

(* ---- med_47.st ---- *)
FUNCTION_BLOCK WindowCleaningSystem
VAR_INPUT
    StartButton : BOOL;
    EmergencyStop : BOOL;
    UpperLimit : BOOL;
    LowerLimit : BOOL;
END_VAR

VAR_OUTPUT
    ElevatorUp : BOOL;
    ElevatorDown : BOOL;
    RotateClockwise : BOOL;
    WaterPump : BOOL;
END_VAR

VAR
    CleaningInProgress : BOOL;
    AtUpperLimitFlag : BOOL;
    DescendingPhase : BOOL;
END_VAR

(* Safety and State Management Logic *)
IF EmergencyStop THEN
    CleaningInProgress := FALSE;
    AtUpperLimitFlag := FALSE;
    DescendingPhase := FALSE;
END_IF;

(* Main Process Sequencing *)
IF NOT EmergencyStop THEN
    (* Start Command Latching *)
    IF StartButton AND NOT CleaningInProgress AND NOT LowerLimit THEN
        CleaningInProgress := TRUE;
        AtUpperLimitFlag := FALSE;
        DescendingPhase := FALSE;
    END_IF;

    (* State: Moving Up to Upper Limit *)
    IF CleaningInProgress AND NOT AtUpperLimitFlag AND NOT DescendingPhase THEN
        IF NOT UpperLimit THEN
            ElevatorUp := TRUE;
            ElevatorDown := FALSE;
            RotateClockwise := FALSE;
            WaterPump := FALSE;
        ELSE
            (* Reached Upper Limit *)
            ElevatorUp := FALSE;
            AtUpperLimitFlag := TRUE;
            DescendingPhase := TRUE;
        END_IF;
    END_IF;

    (* State: Descending and Cleaning *)
    IF CleaningInProgress AND DescendingPhase THEN
        IF NOT LowerLimit THEN
            ElevatorUp := FALSE;
            ElevatorDown := TRUE;
            RotateClockwise := TRUE;
            WaterPump := TRUE;
        ELSE
            (* Reached Lower Limit - Process Complete *)
            ElevatorDown := FALSE;
            RotateClockwise := FALSE;
            WaterPump := FALSE;
            CleaningInProgress := FALSE;
            AtUpperLimitFlag := FALSE;
            DescendingPhase := FALSE;
        END_IF;
    END_IF;

    (* Idle State Outputs *)
    IF NOT CleaningInProgress THEN
        ElevatorUp := FALSE;
        ElevatorDown := FALSE;
        RotateClockwise := FALSE;
        WaterPump := FALSE;
    END_IF;
ELSE
    (* Emergency Stop Active - Force all outputs FALSE *)
    ElevatorUp := FALSE;
    ElevatorDown := FALSE;
    RotateClockwise := FALSE;
    WaterPump := FALSE;
END_IF;

END_FUNCTION_BLOCK

(* ---- med_48.st ---- *)
FUNCTION_BLOCK ChargingStationControl
VAR_INPUT
    EVConnected : BOOL;
    EVVoltage : REAL;
    EVCurrent : REAL;
    EVStateOfCharge : REAL;
    ChargingTimer : TIME;
    MinimumVoltage : REAL;
    MaximumCurrent : REAL;
    MinimumSOC : REAL;
    ChargingVoltage : REAL;
    ChargingCurrent : REAL;
    MaximumChargingTime : TIME;
END_VAR

VAR_OUTPUT
    EVCharging : BOOL;
END_VAR

VAR
    bStartConditionsMet : BOOL;
    bStopConditionsMet : BOOL;
END_VAR

(* Check if all start conditions are met *)
bStartConditionsMet := EVConnected
    AND (EVVoltage > MinimumVoltage)
    AND (EVCurrent <= MaximumCurrent)
    AND (EVStateOfCharge < 100.0)
    AND (ChargingTimer <= MaximumChargingTime);

(* Check if any stop condition is met *)
bStopConditionsMet := (NOT EVConnected)
    OR (EVVoltage <= MinimumVoltage)
    OR (EVCurrent > MaximumCurrent)
    OR (EVStateOfCharge >= 100.0)
    OR (ChargingTimer > MaximumChargingTime);

(* Control charging output *)
IF bStartConditionsMet AND NOT bStopConditionsMet THEN
    EVCharging := TRUE;
ELSE
    EVCharging := FALSE;
END_IF;

END_FUNCTION_BLOCK

(* ---- med_49.st ---- *)
FUNCTION_BLOCK SmartHVACSystem
VAR_INPUT
    TemperatureSensor : REAL; (* Temperature sensor reading *)
    HumiditySensor : REAL; (* Humidity sensor reading *)
END_VAR
VAR_OUTPUT
    HVACMode : INT := 0; (* HVAC operating mode: 0=Off, 1=Cooling, 2=Heating, 3=Ventilation *)
    HVACFanSpeed : INT := 0; (* Fan speed: 0=Off, 1=Low, 2=Medium, 3=High *)
END_VAR
VAR
    DesiredTemperature : REAL := 24.0; (* Desired temperature setting *)
    DesiredHumidity : REAL := 50.0; (* Desired humidity setting *)
    TemperatureThreshold : REAL := 1.0; (* Temperature tolerance threshold *)
    HumidityThreshold : REAL := 5.0; (* Humidity tolerance threshold *)
    AdjustedHumidity : REAL; (* Sanitized humidity input *)
    AdjustedTemperature : REAL; (* Sanitized temperature input *)
    NeedsVentilation : BOOL; (* Flag for ventilation requirement *)
    NeedsHeating : BOOL; (* Flag for heating requirement *)
    NeedsCooling : BOOL; (* Flag for cooling requirement *)
END_VAR

(* Input Sanitization *)
IF HumiditySensor < 0.0 THEN
    AdjustedHumidity := 0.0;
ELSIF HumiditySensor > 100.0 THEN
    AdjustedHumidity := 100.0;
ELSE
    AdjustedHumidity := HumiditySensor;
END_IF;

IF TemperatureSensor < -50.0 THEN
    AdjustedTemperature := -50.0;
ELSIF TemperatureSensor > 100.0 THEN
    AdjustedTemperature := 100.0;
ELSE
    AdjustedTemperature := TemperatureSensor;
END_IF;

(* Determine System Requirements *)
NeedsVentilation := AdjustedHumidity < (DesiredHumidity - HumidityThreshold);
NeedsHeating := AdjustedTemperature < (DesiredTemperature - TemperatureThreshold);
NeedsCooling := AdjustedTemperature > (DesiredTemperature + TemperatureThreshold);

(* Control Logic with Priority: Heating > Cooling > Ventilation *)
IF NeedsHeating THEN
    HVACMode := 2;
    HVACFanSpeed := 3;
ELSIF NeedsCooling THEN
    HVACMode := 1;
    HVACFanSpeed := 3;
ELSIF NeedsVentilation THEN
    HVACMode := 3;
    HVACFanSpeed := 3;
ELSE
    HVACMode := 0;
    HVACFanSpeed := 0;
END_IF;

END_FUNCTION_BLOCK

(* ---- med_50.st ---- *)
FUNCTION_BLOCK CarParkingSystem
VAR_INPUT
    NewCarSlot : INT; (* Input for new car arrival slot number *)
END_VAR
VAR_OUTPUT
    Elevator1Busy : BOOL; (* Elevator 1 status - busy or idle *)
    Elevator2Busy : BOOL; (* Elevator 2 status - busy or idle *)
    Elevator1Position : INT; (* Elevator 1 current position *)
    Elevator2Position : INT; (* Elevator 2 current position *)
END_VAR
VAR
    Elevator1Target : INT; (* Elevator 1 target floor *)
    Elevator2Target : INT; (* Elevator 2 target floor *)
    CarSlots : ARRAY[1..100] OF BOOL; (* Array to represent parking slots - TRUE if occupied *)
    CurrentSlot : INT; (* Loop counter for scanning slots *)
    Elevator1Moving : BOOL; (* Internal flag for elevator 1 movement *)
    Elevator2Moving : BOOL; (* Internal flag for elevator 2 movement *)
    Initialized : BOOL := FALSE; (* System initialization flag *)
END_VAR

(* System initialization - runs once *)
IF NOT Initialized THEN
    FOR CurrentSlot := 1 TO 100 DO
        CarSlots[CurrentSlot] := FALSE;
    END_FOR;
    Elevator1Target := 0;
    Elevator2Target := 0;
    Elevator1Position := 0;
    Elevator2Position := 0;
    Elevator1Busy := FALSE;
    Elevator2Busy := FALSE;
    Elevator1Moving := FALSE;
    Elevator2Moving := FALSE;
    Initialized := TRUE;
END_IF;

(* Process new car arrival *)
IF (NewCarSlot >= 1) AND (NewCarSlot <= 100) THEN
    IF NOT CarSlots[NewCarSlot] THEN
        CarSlots[NewCarSlot] := TRUE;

        (* Assign to appropriate elevator based on slot range *)
        IF (NewCarSlot <= 50) AND NOT Elevator1Busy THEN
            Elevator1Target := NewCarSlot;
            Elevator1Busy := TRUE;
            Elevator1Moving := TRUE;
        ELSIF (NewCarSlot >= 51) AND NOT Elevator2Busy THEN
            Elevator2Target := NewCarSlot;
            Elevator2Busy := TRUE;
            Elevator2Moving := TRUE;
        END_IF;
    END_IF;
END_IF;

(* Elevator 1 movement control *)
IF Elevator1Moving THEN
    IF Elevator1Position < Elevator1Target THEN
        Elevator1Position := Elevator1Position + 1;
    ELSIF Elevator1Position > Elevator1Target THEN
        Elevator1Position := Elevator1Position - 1;
    ELSE
        (* Reached target *)
        Elevator1Moving := FALSE;
        Elevator1Busy := FALSE;
    END_IF;
END_IF;

(* Elevator 2 movement control *)
IF Elevator2Moving THEN
    IF Elevator2Position < Elevator2Target THEN
        Elevator2Position := Elevator2Position + 1;
    ELSIF Elevator2Position > Elevator2Target THEN
        Elevator2Position := Elevator2Position - 1;
    ELSE
        (* Reached target *)
        Elevator2Moving := FALSE;
        Elevator2Busy := FALSE;
    END_IF;
END_IF;

(* Idle elevator scanning for new arrivals - Elevator 1 scans slots 1-50 *)
IF NOT Elevator1Busy THEN
    FOR CurrentSlot := 1 TO 50 DO
        IF CarSlots[CurrentSlot] THEN
            Elevator1Target := CurrentSlot;
            Elevator1Busy := TRUE;
            Elevator1Moving := TRUE;
            EXIT;
        END_IF;
    END_FOR;
END_IF;

(* Idle elevator scanning for new arrivals - Elevator 2 scans slots 51-100 *)
IF NOT Elevator2Busy THEN
    FOR CurrentSlot := 51 TO 100 DO
        IF CarSlots[CurrentSlot] THEN
            Elevator2Target := CurrentSlot;
            Elevator2Busy := TRUE;
            Elevator2Moving := TRUE;
            EXIT;
        END_IF;
    END_FOR;
END_IF;

END_FUNCTION_BLOCK
